LIN {X 0,Y 523.962,Z 330.22,A -85,B 0,C 180,E1 -4900.135,E2 -4900.135} C_VEL
LIN {X 0,Y 523.916,Z 330.218,A -85,B 0,C 180,E1 -4903.168,E2 -4903.168} C_VEL
LIN {X 0,Y 523.936,Z 330.219,A -85,B 0,C 180,E1 -4905.773,E2 -4905.773} C_VEL
LIN {X 0,Y 523.917,Z 330.219,A -85,B 0,C 180,E1 -4906.932,E2 -4906.932} C_VEL
LIN {X 0,Y 523.251,Z 330.304,A -85,B 0,C 180,E1 -4907.573,E2 -4907.573} C_VEL
LIN {X 0,Y 520.406,Z 330.664,A -85,B 0,C 180,E1 -4908.615,E2 -4908.615} C_VEL
LIN {X 0,Y 518,Z 330.967,A -85,B 0,C 180,E1 -4909.454,E2 -4909.454} C_VEL
LIN {X 0,Y 516.963,Z 331.094,A -85,B 0,C 180,E1 -4910.101,E2 -4910.101} C_VEL
LIN {X 0,Y 516.877,Z 331.101,A -85,B 0,C 180,E1 -4910.321,E2 -4910.321} C_VEL
LIN {X 0,Y 516.882,Z 331.095,A -85,B 0,C 180,E1 -4913.343,E2 -4913.343} C_VEL
LIN {X 0,Y 516.909,Z 331.099,A -85,B 0,C 180,E1 -4916.122,E2 -4916.122} C_VEL
LIN {X 0,Y 516.892,Z 331.093,A -85,B 0,C 180,E1 -4918.936,E2 -4918.936} C_VEL
LIN {X 0,Y 516.925,Z 331.093,A -85,B 0,C 180,E1 -4921.586,E2 -4921.586} C_VEL
LIN {X 0,Y 516.934,Z 331.093,A -85,B 0,C 180,E1 -4924.212,E2 -4924.212} C_VEL
LIN {X 0,Y 516.873,Z 331.096,A -85,B 0,C 180,E1 -4926.777,E2 -4926.777} C_VEL
LIN {X 0,Y 516.941,Z 331.095,A -85,B 0,C 180,E1 -4929.732,E2 -4929.732} C_VEL
LIN {X 0,Y 516.931,Z 331.089,A -85,B 0,C 180,E1 -4932.597,E2 -4932.597} C_VEL
LIN {X 0,Y 516.944,Z 331.088,A -85,B 0,C 180,E1 -4935.031,E2 -4935.031} C_VEL
LIN {X 0,Y 516.968,Z 331.086,A -85,B 0,C 180,E1 -4938.234,E2 -4938.234} C_VEL
LIN {X 0,Y 516.973,Z 331.089,A -85,B 0,C 180,E1 -4941.4,E2 -4941.4} C_VEL
LIN {X 0,Y 517.018,Z 331.085,A -85,B 0,C 180,E1 -4943.757,E2 -4943.757} C_VEL
LIN {X 0,Y 517.089,Z 331.077,A -85,B 0,C 180,E1 -4947.663,E2 -4947.663} C_VEL
LIN {X 0,Y 517.097,Z 331.068,A -85,B 0,C 180,E1 -4950.779,E2 -4950.779} C_VEL
LIN {X 0,Y 517.017,Z 331.082,A -85,B 0,C 180,E1 -4953.117,E2 -4953.117} C_VEL
LIN {X 0,Y 517.006,Z 331.08,A -85,B 0,C 180,E1 -4956.243,E2 -4956.243} C_VEL
LIN {X 0,Y 516.955,Z 331.095,A -85,B 0,C 180,E1 -4959.389,E2 -4959.389} C_VEL
LIN {X 0,Y 516.955,Z 331.089,A -85,B 0,C 180,E1 -4961.807,E2 -4961.807} C_VEL
LIN {X 0,Y 516.947,Z 331.093,A -85,B 0,C 180,E1 -4965.146,E2 -4965.146} C_VEL
LIN {X 0,Y 516.928,Z 331.089,A -85,B 0,C 180,E1 -4968.222,E2 -4968.222} C_VEL
LIN {X 0,Y 516.914,Z 331.093,A -85,B 0,C 180,E1 -4970.701,E2 -4970.701} C_VEL
LIN {X 0,Y 516.912,Z 331.091,A -85,B 0,C 180,E1 -4974.071,E2 -4974.071} C_VEL
LIN {X 0,Y 516.93,Z 331.091,A -85,B 0,C 180,E1 -4976.657,E2 -4976.657} C_VEL
LIN {X 0,Y 516.911,Z 331.095,A -85,B 0,C 180,E1 -4979.523,E2 -4979.523} C_VEL
LIN {X 0,Y 516.9,Z 331.094,A -85,B 0,C 180,E1 -4982.544,E2 -4982.544} C_VEL
LIN {X 0,Y 516.882,Z 331.1,A -85,B 0,C 180,E1 -4985.332,E2 -4985.332} C_VEL
LIN {X 0,Y 516.883,Z 331.095,A -85,B 0,C 180,E1 -4987.943,E2 -4987.943} C_VEL
LIN {X 0,Y 516.905,Z 331.099,A -85,B 0,C 180,E1 -4990.738,E2 -4990.738} C_VEL
LIN {X 0,Y 516.879,Z 331.098,A -85,B 0,C 180,E1 -4993.902,E2 -4993.902} C_VEL
LIN {X 0,Y 516.878,Z 331.099,A -85,B 0,C 180,E1 -4996.106,E2 -4996.106} C_VEL
LIN {X 0,Y 516.976,Z 331.211,A -85,B 0,C 180,E1 -4998.813,E2 -4998.813} C_VEL
LIN {X 0,Y 517.149,Z 332.196,A -85,B 0,C 180,E1 -4998.951,E2 -4998.951} C_VEL
LIN {X 0,Y 518.369,Z 337.455,A -85,B 0,C 180,E1 -4999.243,E2 -4999.243} C_VEL
LIN {X 0,Y 518.098,Z 348.894,A -85,B 0,C 180,E1 -4999.884,E2 -4999.884} C_VEL
LIN {X 0,Y 517.795,Z 359.988,A -85,B 0,C 180,E1 -5000.682,E2 -5000.682} C_VEL
LIN {X 0,Y 517.565,Z 369.47,A -85,B 0,C 180,E1 -5001.529,E2 -5001.529} C_VEL
LIN {X 0,Y 517.23,Z 378.856,A -85,B 0,C 180,E1 -5002.551,E2 -5002.551} C_VEL
LIN {X 0,Y 517.051,Z 386.171,A -85,B 0,C 180,E1 -5003.531,E2 -5003.531} C_VEL
LIN {X 0,Y 516.817,Z 393.185,A -85,B 0,C 180,E1 -5004.676,E2 -5004.676} C_VEL
LIN {X 0,Y 516.705,Z 398.028,A -85,B 0,C 180,E1 -5005.635,E2 -5005.635} C_VEL
LIN {X 0,Y 516.538,Z 403.624,A -85,B 0,C 180,E1 -5007.027,E2 -5007.027} C_VEL
LIN {X 0,Y 516.496,Z 407.58,A -85,B 0,C 180,E1 -5008.408,E2 -5008.408} C_VEL
LIN {X 0,Y 516.427,Z 410.24,A -85,B 0,C 180,E1 -5009.766,E2 -5009.766} C_VEL
LIN {X 0,Y 516.38,Z 411.277,A -85,B 0,C 180,E1 -5010.662,E2 -5010.662} C_VEL
LIN {X 0,Y 516.384,Z 411.94,A -85,B 0,C 180,E1 -5012.206,E2 -5012.206} C_VEL
LIN {X 0,Y 516.38,Z 411.461,A -85,B 0,C 180,E1 -5013.312,E2 -5013.312} C_VEL
LIN {X 0,Y 516.426,Z 410.54,A -85,B 0,C 180,E1 -5014.184,E2 -5014.184} C_VEL
LIN {X 0,Y 516.469,Z 409.129,A -85,B 0,C 180,E1 -5015.049,E2 -5015.049} C_VEL
LIN {X 0,Y 516.557,Z 406.079,A -85,B 0,C 180,E1 -5016.337,E2 -5016.337} C_VEL
LIN {X 0,Y 516.692,Z 401.665,A -85,B 0,C 180,E1 -5017.654,E2 -5017.654} C_VEL
LIN {X 0,Y 516.837,Z 395.319,A -85,B 0,C 180,E1 -5019.087,E2 -5019.087} C_VEL
LIN {X 0,Y 517.055,Z 388.019,A -85,B 0,C 180,E1 -5020.342,E2 -5020.342} C_VEL
LIN {X 0,Y 517.297,Z 380.58,A -85,B 0,C 180,E1 -5021.381,E2 -5021.381} C_VEL
LIN {X 0,Y 517.573,Z 371.1,A -85,B 0,C 180,E1 -5022.457,E2 -5022.457} C_VEL
LIN {X 0,Y 517.845,Z 361.431,A -85,B 0,C 180,E1 -5023.339,E2 -5023.339} C_VEL
LIN {X 0,Y 518.133,Z 350.286,A -85,B 0,C 180,E1 -5024.158,E2 -5024.158} C_VEL
LIN {X 0,Y 518.394,Z 338.832,A -85,B 0,C 180,E1 -5024.816,E2 -5024.816} C_VEL
LIN {X 0,Y 518.185,Z 335.842,A -85,B 0,C 180,E1 -5024.968,E2 -5024.968} C_VEL
LIN {X 0,Y 517.053,Z 331.596,A -85,B 0,C 180,E1 -5025.235,E2 -5025.235} C_VEL
LIN {X 0,Y 516.923,Z 331.103,A -85,B 0,C 180,E1 -5025.432,E2 -5025.432} C_VEL
LIN {X 0,Y 516.955,Z 331.09,A -85,B 0,C 180,E1 -5028.233,E2 -5028.233} C_VEL
LIN {X 0,Y 516.958,Z 331.095,A -85,B 0,C 180,E1 -5031.4,E2 -5031.4} C_VEL
LIN {X 0,Y 516.989,Z 331.087,A -85,B 0,C 180,E1 -5033.757,E2 -5033.757} C_VEL
LIN {X 0,Y 517.001,Z 331.085,A -85,B 0,C 180,E1 -5036.883,E2 -5036.883} C_VEL
LIN {X 0,Y 517.068,Z 331.074,A -85,B 0,C 180,E1 -5040,E2 -5040} C_VEL
LIN {X 0,Y 517.002,Z 331.088,A -85,B 0,C 180,E1 -5043.117,E2 -5043.117} C_VEL
LIN {X 0,Y 516.989,Z 331.082,A -85,B 0,C 180,E1 -5046.243,E2 -5046.243} C_VEL
LIN {X 0,Y 516.936,Z 331.094,A -85,B 0,C 180,E1 -5049.39,E2 -5049.39} C_VEL
LIN {X 0,Y 516.941,Z 331.089,A -85,B 0,C 180,E1 -5051.807,E2 -5051.807} C_VEL
LIN {X 0,Y 516.933,Z 331.097,A -85,B 0,C 180,E1 -5055.147,E2 -5055.147} C_VEL
LIN {X 0,Y 516.905,Z 331.091,A -85,B 0,C 180,E1 -5058.223,E2 -5058.223} C_VEL
LIN {X 0,Y 516.901,Z 331.097,A -85,B 0,C 180,E1 -5060.702,E2 -5060.702} C_VEL
LIN {X 0,Y 516.879,Z 331.095,A -85,B 0,C 180,E1 -5064.074,E2 -5064.074} C_VEL
LIN {X 0,Y 516.914,Z 331.096,A -85,B 0,C 180,E1 -5066.659,E2 -5066.659} C_VEL
LIN {X 0,Y 516.899,Z 331.095,A -85,B 0,C 180,E1 -5069.524,E2 -5069.524} C_VEL
LIN {X 0,Y 516.885,Z 331.1,A -85,B 0,C 180,E1 -5072.544,E2 -5072.544} C_VEL
LIN {X 0,Y 516.857,Z 331.102,A -85,B 0,C 180,E1 -5075.33,E2 -5075.33} C_VEL
LIN {X 0,Y 516.871,Z 331.098,A -85,B 0,C 180,E1 -5077.943,E2 -5077.943} C_VEL
LIN {X 0,Y 516.846,Z 331.108,A -85,B 0,C 180,E1 -5080.745,E2 -5080.745} C_VEL
LIN {X 0,Y 516.875,Z 331.098,A -85,B 0,C 180,E1 -5083.904,E2 -5083.904} C_VEL
LIN {X 0,Y 516.875,Z 331.1,A -85,B 0,C 180,E1 -5086.108,E2 -5086.108} C_VEL
LIN {X 0,Y 516.849,Z 331.104,A -85,B 0,C 180,E1 -5089.256,E2 -5089.256} C_VEL
LIN {X 0,Y 516.911,Z 331.323,A -85,B 0,C 180,E1 -5092.053,E2 -5092.053} C_VEL
LIN {X 0,Y 518.241,Z 338.355,A -85,B 0,C 180,E1 -5093.85,E2 -5093.85} C_VEL
LIN {X 0,Y 518.188,Z 344.44,A -85,B 0,C 180,E1 -5095.277,E2 -5095.277} C_VEL
LIN {X 0,Y 517.75,Z 358.665,A -85,B 0,C 180,E1 -5098.45,E2 -5098.45} C_VEL
LIN {X 0,Y 517.637,Z 370.384,A -85,B 0,C 180,E1 -5100.963,E2 -5100.963} C_VEL
LIN {X 0,Y 517.472,Z 384.841,A -85,B 0,C 180,E1 -5103.959,E2 -5103.959} C_VEL
LIN {X 0,Y 517.305,Z 400.935,A -85,B 0,C 180,E1 -5107.195,E2 -5107.195} C_VEL
LIN {X 0,Y 517.105,Z 416.945,A -85,B 0,C 180,E1 -5110.344,E2 -5110.344} C_VEL
LIN {X 0,Y 516.951,Z 430.617,A -85,B 0,C 180,E1 -5113.005,E2 -5113.005} C_VEL
LIN {X 0,Y 516.782,Z 445.74,A -85,B 0,C 180,E1 -5115.931,E2 -5115.931} C_VEL
LIN {X 0,Y 516.772,Z 446.824,A -85,B 0,C 180,E1 -5116.056,E2 -5116.056} C_VEL
LIN {X 0,Y 518.022,Z 457.401,A -85,B 0,C 180,E1 -5116.316,E2 -5116.316} C_VEL
LIN {X 0,Y 518.329,Z 462.091,A -85,B 0,C 180,E1 -5116.449,E2 -5116.449} C_VEL
LIN {X 0,Y 518.085,Z 475.478,A -85,B 0,C 180,E1 -5116.917,E2 -5116.917} C_VEL
LIN {X 0,Y 517.828,Z 488.026,A -85,B 0,C 180,E1 -5117.532,E2 -5117.532} C_VEL
LIN {X 0,Y 517.576,Z 499.386,A -85,B 0,C 180,E1 -5118.248,E2 -5118.248} C_VEL
LIN {X 0,Y 517.292,Z 510.601,A -85,B 0,C 180,E1 -5119.135,E2 -5119.135} C_VEL
LIN {X 0,Y 516.965,Z 519.69,A -85,B 0,C 180,E1 -5120.019,E2 -5120.019} C_VEL
LIN {X 0,Y 516.735,Z 529.581,A -85,B 0,C 180,E1 -5121.199,E2 -5121.199} C_VEL
LIN {X 0,Y 516.563,Z 537.519,A -85,B 0,C 180,E1 -5122.377,E2 -5122.377} C_VEL
LIN {X 0,Y 516.462,Z 543.17,A -85,B 0,C 180,E1 -5123.406,E2 -5123.406} C_VEL
LIN {X 0,Y 516.403,Z 548.195,A -85,B 0,C 180,E1 -5124.533,E2 -5124.533} C_VEL
LIN {X 0,Y 516.36,Z 552.279,A -85,B 0,C 180,E1 -5125.707,E2 -5125.707} C_VEL
LIN {X 0,Y 516.282,Z 555.285,A -85,B 0,C 180,E1 -5126.879,E2 -5126.879} C_VEL
LIN {X 0,Y 516.261,Z 556.726,A -85,B 0,C 180,E1 -5127.659,E2 -5127.659} C_VEL
LIN {X 0,Y 516.162,Z 558.361,A -85,B 0,C 180,E1 -5129.22,E2 -5129.22} C_VEL
LIN {X 0,Y 516.159,Z 558.584,A -85,B 0,C 180,E1 -5130,E2 -5130} C_VEL
LIN {X 0,Y 516.162,Z 558.364,A -85,B 0,C 180,E1 -5130.78,E2 -5130.78} C_VEL
LIN {X 0,Y 516.261,Z 556.735,A -85,B 0,C 180,E1 -5132.341,E2 -5132.341} C_VEL
LIN {X 0,Y 516.282,Z 555.301,A -85,B 0,C 180,E1 -5133.121,E2 -5133.121} C_VEL
LIN {X 0,Y 516.36,Z 552.302,A -85,B 0,C 180,E1 -5134.293,E2 -5134.293} C_VEL
LIN {X 0,Y 516.403,Z 548.232,A -85,B 0,C 180,E1 -5135.467,E2 -5135.467} C_VEL
LIN {X 0,Y 516.483,Z 542.141,A -85,B 0,C 180,E1 -5136.805,E2 -5136.805} C_VEL
LIN {X 0,Y 516.64,Z 535.153,A -85,B 0,C 180,E1 -5138.015,E2 -5138.015} C_VEL
LIN {X 0,Y 516.813,Z 526.702,A -85,B 0,C 180,E1 -5139.194,E2 -5139.194} C_VEL
LIN {X 0,Y 517.04,Z 518.021,A -85,B 0,C 180,E1 -5140.178,E2 -5140.178} C_VEL
LIN {X 0,Y 517.339,Z 507.38,A -85,B 0,C 180,E1 -5141.162,E2 -5141.162} C_VEL
LIN {X 0,Y 517.652,Z 496.773,A -85,B 0,C 180,E1 -5141.956,E2 -5141.956} C_VEL
LIN {X 0,Y 517.883,Z 485.3,A -85,B 0,C 180,E1 -5142.64,E2 -5142.64} C_VEL
LIN {X 0,Y 518.196,Z 472.203,A -85,B 0,C 180,E1 -5143.23,E2 -5143.23} C_VEL
LIN {X 0,Y 518.357,Z 459.09,A -85,B 0,C 180,E1 -5143.65,E2 -5143.65} C_VEL
LIN {X 0,Y 516.789,Z 447.402,A -85,B 0,C 180,E1 -5143.943,E2 -5143.943} C_VEL
LIN {X 0,Y 516.83,Z 445.814,A -85,B 0,C 180,E1 -5144.168,E2 -5144.168} C_VEL
LIN {X 0,Y 516.996,Z 429.457,A -85,B 0,C 180,E1 -5147.401,E2 -5147.401} C_VEL
LIN {X 0,Y 517.162,Z 415.971,A -85,B 0,C 180,E1 -5150.1,E2 -5150.1} C_VEL
LIN {X 0,Y 517.433,Z 402.623,A -85,B 0,C 180,E1 -5152.821,E2 -5152.821} C_VEL
LIN {X 0,Y 517.748,Z 387.104,A -85,B 0,C 180,E1 -5156.064,E2 -5156.064} C_VEL
LIN {X 0,Y 518.026,Z 372.315,A -85,B 0,C 180,E1 -5159.235,E2 -5159.235} C_VEL
LIN {X 0,Y 518.311,Z 360.147,A -85,B 0,C 180,E1 -5161.925,E2 -5161.925} C_VEL
LIN {X 0,Y 518.941,Z 344.977,A -85,B 0,C 180,E1 -5165.376,E2 -5165.376} C_VEL
LIN {X 0,Y 518.836,Z 340.922,A -85,B 0,C 180,E1 -5166.342,E2 -5166.342} C_VEL
LIN {X 0,Y 516.875,Z 331.191,A -85,B 0,C 180,E1 -5168.864,E2 -5168.864} C_VEL
LIN {X 0,Y 516.878,Z 331.103,A -85,B 0,C 180,E1 -5171.777,E2 -5171.777} C_VEL
LIN {X 0,Y 516.89,Z 331.1,A -85,B 0,C 180,E1 -5175.006,E2 -5175.006} C_VEL
LIN {X 0,Y 516.88,Z 331.095,A -85,B 0,C 180,E1 -5178.401,E2 -5178.401} C_VEL
LIN {X 0,Y 516.869,Z 331.105,A -85,B 0,C 180,E1 -5181.283,E2 -5181.283} C_VEL
LIN {X 0,Y 516.862,Z 331.097,A -85,B 0,C 180,E1 -5184.219,E2 -5184.219} C_VEL
LIN {X 0,Y 516.872,Z 331.102,A -85,B 0,C 180,E1 -5187.051,E2 -5187.051} C_VEL
LIN {X 0,Y 516.877,Z 331.097,A -85,B 0,C 180,E1 -5189.795,E2 -5189.795} C_VEL
LIN {X 0,Y 516.915,Z 331.091,A -85,B 0,C 180,E1 -5192.467,E2 -5192.467} C_VEL
LIN {X 0,Y 516.861,Z 331.105,A -85,B 0,C 180,E1 -5195.069,E2 -5195.069} C_VEL
LIN {X 0,Y 516.859,Z 331.1,A -85,B 0,C 180,E1 -5197.621,E2 -5197.621} C_VEL
LIN {X 0,Y 516.92,Z 331.09,A -85,B 0,C 180,E1 -5200.129,E2 -5200.129} C_VEL
LIN {X 0,Y 516.896,Z 331.096,A -85,B 0,C 180,E1 -5202.595,E2 -5202.595} C_VEL
LIN {X 0,Y 516.931,Z 331.098,A -85,B 0,C 180,E1 -5205.03,E2 -5205.03} C_VEL
LIN {X 0,Y 516.955,Z 331.086,A -85,B 0,C 180,E1 -5208.233,E2 -5208.233} C_VEL
LIN {X 0,Y 516.945,Z 331.089,A -85,B 0,C 180,E1 -5211.399,E2 -5211.399} C_VEL
LIN {X 0,Y 516.989,Z 331.081,A -85,B 0,C 180,E1 -5213.757,E2 -5213.757} C_VEL
LIN {X 0,Y 517.001,Z 331.089,A -85,B 0,C 180,E1 -5216.883,E2 -5216.883} C_VEL
LIN {X 0,Y 517.068,Z 331.072,A -85,B 0,C 180,E1 -5220,E2 -5220} C_VEL
LIN {X 0,Y 517.001,Z 331.084,A -85,B 0,C 180,E1 -5223.117,E2 -5223.117} C_VEL
LIN {X 0,Y 516.989,Z 331.084,A -85,B 0,C 180,E1 -5226.243,E2 -5226.243} C_VEL
LIN {X 0,Y 516.943,Z 331.088,A -85,B 0,C 180,E1 -5229.389,E2 -5229.389} C_VEL
LIN {X 0,Y 516.943,Z 331.087,A -85,B 0,C 180,E1 -5231.808,E2 -5231.808} C_VEL
LIN {X 0,Y 516.936,Z 331.09,A -85,B 0,C 180,E1 -5235.148,E2 -5235.148} C_VEL
LIN {X 0,Y 516.915,Z 331.095,A -85,B 0,C 180,E1 -5238.223,E2 -5238.223} C_VEL
LIN {X 0,Y 516.906,Z 331.098,A -85,B 0,C 180,E1 -5240.702,E2 -5240.702} C_VEL
LIN {X 0,Y 516.883,Z 331.095,A -85,B 0,C 180,E1 -5243.223,E2 -5243.223} C_VEL
LIN {X 0,Y 516.934,Z 331.094,A -85,B 0,C 180,E1 -5246.197,E2 -5246.197} C_VEL
LIN {X 0,Y 516.928,Z 331.089,A -85,B 0,C 180,E1 -5249.304,E2 -5249.304} C_VEL
LIN {X 0,Y 516.889,Z 331.1,A -85,B 0,C 180,E1 -5252.544,E2 -5252.544} C_VEL
LIN {X 0,Y 516.872,Z 331.096,A -85,B 0,C 180,E1 -5255.332,E2 -5255.332} C_VEL
LIN {X 0,Y 516.874,Z 331.1,A -85,B 0,C 180,E1 -5257.944,E2 -5257.944} C_VEL
LIN {X 0,Y 516.898,Z 331.095,A -85,B 0,C 180,E1 -5260.74,E2 -5260.74} C_VEL
LIN {X 0,Y 516.877,Z 331.1,A -85,B 0,C 180,E1 -5263.904,E2 -5263.904} C_VEL
LIN {X 0,Y 516.878,Z 331.104,A -85,B 0,C 180,E1 -5266.108,E2 -5266.108} C_VEL
LIN {X 0,Y 516.911,Z 331.096,A -85,B 0,C 180,E1 -5268.399,E2 -5268.399} C_VEL
LIN {X 0,Y 516.877,Z 331.101,A -85,B 0,C 180,E1 -5270.321,E2 -5270.321} C_VEL
LIN {X 0,Y 516.207,Z 331.181,A -85,B 0,C 180,E1 -5270.971,E2 -5270.971} C_VEL
LIN {X 0,Y 513.361,Z 331.542,A -85,B 0,C 180,E1 -5272.027,E2 -5272.027} C_VEL
LIN {X 0,Y 510.954,Z 331.841,A -85,B 0,C 180,E1 -5272.877,E2 -5272.877} C_VEL
LIN {X 0,Y 509.915,Z 331.966,A -85,B 0,C 180,E1 -5273.534,E2 -5273.534} C_VEL
LIN {X 0,Y 509.827,Z 331.976,A -85,B 0,C 180,E1 -5273.756,E2 -5273.756} C_VEL
LIN {X 0,Y 509.859,Z 331.972,A -85,B 0,C 180,E1 -5276.54,E2 -5276.54} C_VEL
LIN {X 0,Y 509.849,Z 331.972,A -85,B 0,C 180,E1 -5279.335,E2 -5279.335} C_VEL
LIN {X 0,Y 509.896,Z 331.972,A -85,B 0,C 180,E1 -5282.055,E2 -5282.055} C_VEL
LIN {X 0,Y 509.879,Z 331.967,A -85,B 0,C 180,E1 -5284.705,E2 -5284.705} C_VEL
LIN {X 0,Y 509.837,Z 331.976,A -85,B 0,C 180,E1 -5287.456,E2 -5287.456} C_VEL
LIN {X 0,Y 509.918,Z 331.971,A -85,B 0,C 180,E1 -5289.845,E2 -5289.845} C_VEL
LIN {X 0,Y 509.887,Z 331.968,A -85,B 0,C 180,E1 -5293.175,E2 -5293.175} C_VEL
LIN {X 0,Y 509.867,Z 331.976,A -85,B 0,C 180,E1 -5295.635,E2 -5295.635} C_VEL
LIN {X 0,Y 509.916,Z 331.963,A -85,B 0,C 180,E1 -5298.875,E2 -5298.875} C_VEL
LIN {X 0,Y 509.955,Z 331.961,A -85,B 0,C 180,E1 -5302.079,E2 -5302.079} C_VEL
LIN {X 0,Y 509.988,Z 331.954,A -85,B 0,C 180,E1 -5304.465,E2 -5304.465} C_VEL
LIN {X 0,Y 510.059,Z 331.953,A -85,B 0,C 180,E1 -5307.631,E2 -5307.631} C_VEL
LIN {X 0,Y 510.067,Z 331.944,A -85,B 0,C 180,E1 -5310.789,E2 -5310.789} C_VEL
LIN {X 0,Y 509.959,Z 331.961,A -85,B 0,C 180,E1 -5313.16,E2 -5313.16} C_VEL
LIN {X 0,Y 509.957,Z 331.957,A -85,B 0,C 180,E1 -5316.33,E2 -5316.33} C_VEL
LIN {X 0,Y 509.918,Z 331.963,A -85,B 0,C 180,E1 -5318.72,E2 -5318.72} C_VEL
LIN {X 0,Y 509.907,Z 331.965,A -85,B 0,C 180,E1 -5321.931,E2 -5321.931} C_VEL
LIN {X 0,Y 509.896,Z 331.973,A -85,B 0,C 180,E1 -5325.241,E2 -5325.241} C_VEL
LIN {X 0,Y 509.891,Z 331.966,A -85,B 0,C 180,E1 -5328.001,E2 -5328.001} C_VEL
LIN {X 0,Y 509.852,Z 331.976,A -85,B 0,C 180,E1 -5331.001,E2 -5331.001} C_VEL
LIN {X 0,Y 509.838,Z 331.976,A -85,B 0,C 180,E1 -5333.562,E2 -5333.562} C_VEL
LIN {X 0,Y 509.914,Z 331.963,A -85,B 0,C 180,E1 -5336.379,E2 -5336.379} C_VEL
LIN {X 0,Y 509.877,Z 331.972,A -85,B 0,C 180,E1 -5338.843,E2 -5338.843} C_VEL
LIN {X 0,Y 509.824,Z 331.976,A -85,B 0,C 180,E1 -5341.589,E2 -5341.589} C_VEL
LIN {X 0,Y 509.853,Z 331.971,A -85,B 0,C 180,E1 -5344.412,E2 -5344.412} C_VEL
LIN {X 0,Y 509.821,Z 331.979,A -85,B 0,C 180,E1 -5347.339,E2 -5347.339} C_VEL
LIN {X 0,Y 509.86,Z 331.973,A -85,B 0,C 180,E1 -5350.379,E2 -5350.379} C_VEL
LIN {X 0,Y 509.837,Z 331.98,A -85,B 0,C 180,E1 -5353.064,E2 -5353.064} C_VEL
LIN {X 0,Y 509.826,Z 331.977,A -85,B 0,C 180,E1 -5355.791,E2 -5355.791} C_VEL
LIN {X 0,Y 509.921,Z 332.178,A -85,B 0,C 180,E1 -5358.649,E2 -5358.649} C_VEL
LIN {X 0,Y 510.142,Z 333.081,A -85,B 0,C 180,E1 -5358.772,E2 -5358.772} C_VEL
LIN {X 0,Y 511.495,Z 338.635,A -85,B 0,C 180,E1 -5359.085,E2 -5359.085} C_VEL
LIN {X 0,Y 511.202,Z 350.173,A -85,B 0,C 180,E1 -5359.747,E2 -5359.747} C_VEL
LIN {X 0,Y 510.893,Z 361.197,A -85,B 0,C 180,E1 -5360.555,E2 -5360.555} C_VEL
LIN {X 0,Y 510.59,Z 371.747,A -85,B 0,C 180,E1 -5361.524,E2 -5361.524} C_VEL
LIN {X 0,Y 510.244,Z 381.905,A -85,B 0,C 180,E1 -5362.696,E2 -5362.696} C_VEL
LIN {X 0,Y 510.001,Z 390.072,A -85,B 0,C 180,E1 -5363.874,E2 -5363.874} C_VEL
LIN {X 0,Y 509.798,Z 396.88,A -85,B 0,C 180,E1 -5365.102,E2 -5365.102} C_VEL
LIN {X 0,Y 509.638,Z 401.649,A -85,B 0,C 180,E1 -5366.172,E2 -5366.172} C_VEL
LIN {X 0,Y 509.491,Z 406.118,A -85,B 0,C 180,E1 -5367.454,E2 -5367.454} C_VEL
LIN {X 0,Y 509.457,Z 409.548,A -85,B 0,C 180,E1 -5368.79,E2 -5368.79} C_VEL
LIN {X 0,Y 509.374,Z 411.996,A -85,B 0,C 180,E1 -5370.367,E2 -5370.367} C_VEL
LIN {X 0,Y 509.358,Z 412.662,A -85,B 0,C 180,E1 -5371.124,E2 -5371.124} C_VEL
LIN {X 0,Y 509.351,Z 412.963,A -85,B 0,C 180,E1 -5372.022,E2 -5372.022} C_VEL
LIN {X 0,Y 509.364,Z 412.736,A -85,B 0,C 180,E1 -5372.914,E2 -5372.914} C_VEL
LIN {X 0,Y 509.381,Z 412.029,A -85,B 0,C 180,E1 -5373.8,E2 -5373.8} C_VEL
LIN {X 0,Y 509.433,Z 410.842,A -85,B 0,C 180,E1 -5374.68,E2 -5374.68} C_VEL
LIN {X 0,Y 509.545,Z 408.16,A -85,B 0,C 180,E1 -5375.991,E2 -5375.991} C_VEL
LIN {X 0,Y 509.671,Z 403.589,A -85,B 0,C 180,E1 -5377.497,E2 -5377.497} C_VEL
LIN {X 0,Y 509.794,Z 399.236,A -85,B 0,C 180,E1 -5378.572,E2 -5378.572} C_VEL
LIN {X 0,Y 509.987,Z 392.761,A -85,B 0,C 180,E1 -5379.848,E2 -5379.848} C_VEL
LIN {X 0,Y 510.265,Z 384.563,A -85,B 0,C 180,E1 -5381.115,E2 -5381.115} C_VEL
LIN {X 0,Y 510.578,Z 375.533,A -85,B 0,C 180,E1 -5382.232,E2 -5382.232} C_VEL
LIN {X 0,Y 510.881,Z 365.729,A -85,B 0,C 180,E1 -5383.209,E2 -5383.209} C_VEL
LIN {X 0,Y 511.193,Z 355.362,A -85,B 0,C 180,E1 -5384.04,E2 -5384.04} C_VEL
LIN {X 0,Y 511.496,Z 344.492,A -85,B 0,C 180,E1 -5384.737,E2 -5384.737} C_VEL
LIN {X 0,Y 511.492,Z 338.239,A -85,B 0,C 180,E1 -5385.071,E2 -5385.071} C_VEL
LIN {X 0,Y 510.002,Z 332.602,A -85,B 0,C 180,E1 -5385.409,E2 -5385.409} C_VEL
LIN {X 0,Y 509.871,Z 331.979,A -85,B 0,C 180,E1 -5385.634,E2 -5385.634} C_VEL
LIN {X 0,Y 509.906,Z 331.97,A -85,B 0,C 180,E1 -5388.874,E2 -5388.874} C_VEL
LIN {X 0,Y 509.94,Z 331.963,A -85,B 0,C 180,E1 -5392.078,E2 -5392.078} C_VEL
LIN {X 0,Y 509.967,Z 331.958,A -85,B 0,C 180,E1 -5394.464,E2 -5394.464} C_VEL
LIN {X 0,Y 510.041,Z 331.953,A -85,B 0,C 180,E1 -5397.631,E2 -5397.631} C_VEL
LIN {X 0,Y 510.04,Z 331.95,A -85,B 0,C 180,E1 -5400,E2 -5400} C_VEL
LIN {X 0,Y 510.039,Z 331.948,A -85,B 0,C 180,E1 -5402.369,E2 -5402.369} C_VEL
LIN {X 0,Y 509.966,Z 331.962,A -85,B 0,C 180,E1 -5405.536,E2 -5405.536} C_VEL
LIN {X 0,Y 509.909,Z 331.964,A -85,B 0,C 180,E1 -5407.922,E2 -5407.922} C_VEL
LIN {X 0,Y 509.901,Z 331.974,A -85,B 0,C 180,E1 -5411.126,E2 -5411.126} C_VEL
LIN {X 0,Y 509.851,Z 331.972,A -85,B 0,C 180,E1 -5414.366,E2 -5414.366} C_VEL
LIN {X 0,Y 509.863,Z 331.976,A -85,B 0,C 180,E1 -5416.826,E2 -5416.826} C_VEL
LIN {X 0,Y 509.906,Z 331.964,A -85,B 0,C 180,E1 -5420.156,E2 -5420.156} C_VEL
LIN {X 0,Y 509.81,Z 331.977,A -85,B 0,C 180,E1 -5423.565,E2 -5423.565} C_VEL
LIN {X 0,Y 509.901,Z 331.966,A -85,B 0,C 180,E1 -5426.379,E2 -5426.379} C_VEL
LIN {X 0,Y 509.863,Z 331.976,A -85,B 0,C 180,E1 -5428.845,E2 -5428.845} C_VEL
LIN {X 0,Y 509.809,Z 331.978,A -85,B 0,C 180,E1 -5431.591,E2 -5431.591} C_VEL
LIN {X 0,Y 509.83,Z 331.978,A -85,B 0,C 180,E1 -5434.415,E2 -5434.415} C_VEL
LIN {X 0,Y 509.808,Z 331.98,A -85,B 0,C 180,E1 -5437.342,E2 -5437.342} C_VEL
LIN {X 0,Y 509.807,Z 331.982,A -85,B 0,C 180,E1 -5440.385,E2 -5440.385} C_VEL
LIN {X 0,Y 509.789,Z 331.985,A -85,B 0,C 180,E1 -5443.06,E2 -5443.06} C_VEL
LIN {X 0,Y 509.816,Z 331.978,A -85,B 0,C 180,E1 -5445.794,E2 -5445.794} C_VEL
LIN {X 0,Y 509.826,Z 331.982,A -85,B 0,C 180,E1 -5448.573,E2 -5448.573} C_VEL
LIN {X 0,Y 509.85,Z 332.132,A -85,B 0,C 180,E1 -5451.787,E2 -5451.787} C_VEL
LIN {X 0,Y 511.288,Z 339.689,A -85,B 0,C 180,E1 -5453.769,E2 -5453.769} C_VEL
LIN {X 0,Y 511.253,Z 345.707,A -85,B 0,C 180,E1 -5455.207,E2 -5455.207} C_VEL
LIN {X 0,Y 510.76,Z 360.437,A -85,B 0,C 180,E1 -5458.552,E2 -5458.552} C_VEL
LIN {X 0,Y 510.6,Z 371.564,A -85,B 0,C 180,E1 -5460.976,E2 -5460.976} C_VEL
LIN {X 0,Y 510.422,Z 385.228,A -85,B 0,C 180,E1 -5463.858,E2 -5463.858} C_VEL
LIN {X 0,Y 510.24,Z 401.062,A -85,B 0,C 180,E1 -5467.101,E2 -5467.101} C_VEL
LIN {X 0,Y 510.012,Z 416.878,A -85,B 0,C 180,E1 -5470.269,E2 -5470.269} C_VEL
LIN {X 0,Y 509.871,Z 430.533,A -85,B 0,C 180,E1 -5472.968,E2 -5472.968} C_VEL
LIN {X 0,Y 509.722,Z 445.31,A -85,B 0,C 180,E1 -5475.834,E2 -5475.834} C_VEL
LIN {X 0,Y 509.904,Z 448.112,A -85,B 0,C 180,E1 -5475.928,E2 -5475.928} C_VEL
LIN {X 0,Y 511.065,Z 458.131,A -85,B 0,C 180,E1 -5476.177,E2 -5476.177} C_VEL
LIN {X 0,Y 511.361,Z 463.388,A -85,B 0,C 180,E1 -5476.337,E2 -5476.337} C_VEL
LIN {X 0,Y 511.066,Z 476.455,A -85,B 0,C 180,E1 -5476.835,E2 -5476.835} C_VEL
LIN {X 0,Y 510.784,Z 488.569,A -85,B 0,C 180,E1 -5477.459,E2 -5477.459} C_VEL
LIN {X 0,Y 510.528,Z 499.598,A -85,B 0,C 180,E1 -5478.184,E2 -5478.184} C_VEL
LIN {X 0,Y 510.21,Z 510.505,A -85,B 0,C 180,E1 -5479.082,E2 -5479.082} C_VEL
LIN {X 0,Y 509.876,Z 520.348,A -85,B 0,C 180,E1 -5480.079,E2 -5480.079} C_VEL
LIN {X 0,Y 509.675,Z 528.458,A -85,B 0,C 180,E1 -5481.076,E2 -5481.076} C_VEL
LIN {X 0,Y 509.513,Z 536.424,A -85,B 0,C 180,E1 -5482.271,E2 -5482.271} C_VEL
LIN {X 0,Y 509.367,Z 543.727,A -85,B 0,C 180,E1 -5483.663,E2 -5483.663} C_VEL
LIN {X 0,Y 509.294,Z 548.604,A -85,B 0,C 180,E1 -5484.854,E2 -5484.854} C_VEL
LIN {X 0,Y 509.336,Z 552.348,A -85,B 0,C 180,E1 -5486.044,E2 -5486.044} C_VEL
LIN {X 0,Y 509.243,Z 554.261,A -85,B 0,C 180,E1 -5486.836,E2 -5486.836} C_VEL
LIN {X 0,Y 509.222,Z 555.711,A -85,B 0,C 180,E1 -5487.627,E2 -5487.627} C_VEL
LIN {X 0,Y 509.156,Z 557.366,A -85,B 0,C 180,E1 -5489.209,E2 -5489.209} C_VEL
LIN {X 0,Y 509.149,Z 557.594,A -85,B 0,C 180,E1 -5490,E2 -5490} C_VEL
LIN {X 0,Y 509.156,Z 557.379,A -85,B 0,C 180,E1 -5490.791,E2 -5490.791} C_VEL
LIN {X 0,Y 509.218,Z 555.753,A -85,B 0,C 180,E1 -5492.373,E2 -5492.373} C_VEL
LIN {X 0,Y 509.237,Z 554.319,A -85,B 0,C 180,E1 -5493.164,E2 -5493.164} C_VEL
LIN {X 0,Y 509.282,Z 551.319,A -85,B 0,C 180,E1 -5494.353,E2 -5494.353} C_VEL
LIN {X 0,Y 509.342,Z 547.251,A -85,B 0,C 180,E1 -5495.543,E2 -5495.543} C_VEL
LIN {X 0,Y 509.415,Z 541.338,A -85,B 0,C 180,E1 -5496.864,E2 -5496.864} C_VEL
LIN {X 0,Y 509.571,Z 534.166,A -85,B 0,C 180,E1 -5498.127,E2 -5498.127} C_VEL
LIN {X 0,Y 509.758,Z 525.708,A -85,B 0,C 180,E1 -5499.323,E2 -5499.323} C_VEL
LIN {X 0,Y 510.009,Z 517.023,A -85,B 0,C 180,E1 -5500.32,E2 -5500.32} C_VEL
LIN {X 0,Y 510.298,Z 506.373,A -85,B 0,C 180,E1 -5501.318,E2 -5501.318} C_VEL
LIN {X 0,Y 510.618,Z 495.923,A -85,B 0,C 180,E1 -5502.112,E2 -5502.112} C_VEL
LIN {X 0,Y 510.909,Z 484.279,A -85,B 0,C 180,E1 -5502.815,E2 -5502.815} C_VEL
LIN {X 0,Y 511.274,Z 471.177,A -85,B 0,C 180,E1 -5503.412,E2 -5503.412} C_VEL
LIN {X 0,Y 511.298,Z 459.401,A -85,B 0,C 180,E1 -5503.804,E2 -5503.804} C_VEL
LIN {X 0,Y 509.774,Z 447.382,A -85,B 0,C 180,E1 -5504.113,E2 -5504.113} C_VEL
LIN {X 0,Y 509.75,Z 445.928,A -85,B 0,C 180,E1 -5504.19,E2 -5504.19} C_VEL
LIN {X 0,Y 509.91,Z 430.664,A -85,B 0,C 180,E1 -5507.237,E2 -5507.237} C_VEL
LIN {X 0,Y 510.085,Z 417.396,A -85,B 0,C 180,E1 -5509.938,E2 -5509.938} C_VEL
LIN {X 0,Y 510.372,Z 404.121,A -85,B 0,C 180,E1 -5512.688,E2 -5512.688} C_VEL
LIN {X 0,Y 510.689,Z 388.957,A -85,B 0,C 180,E1 -5515.908,E2 -5515.908} C_VEL
LIN {X 0,Y 511.01,Z 374.729,A -85,B 0,C 180,E1 -5518.998,E2 -5518.998} C_VEL
LIN {X 0,Y 511.349,Z 361.565,A -85,B 0,C 180,E1 -5521.946,E2 -5521.946} C_VEL
LIN {X 0,Y 511.967,Z 347.435,A -85,B 0,C 180,E1 -5525.207,E2 -5525.207} C_VEL
LIN {X 0,Y 512.052,Z 343.388,A -85,B 0,C 180,E1 -5526.169,E2 -5526.169} C_VEL
LIN {X 0,Y 510.072,Z 333.104,A -85,B 0,C 180,E1 -5528.822,E2 -5528.822} C_VEL
LIN {X 0,Y 509.847,Z 332.053,A -85,B 0,C 180,E1 -5529.16,E2 -5529.16} C_VEL
LIN {X 0,Y 509.825,Z 331.981,A -85,B 0,C 180,E1 -5531.892,E2 -5531.892} C_VEL
LIN {X 0,Y 509.833,Z 331.976,A -85,B 0,C 180,E1 -5534.669,E2 -5534.669} C_VEL
LIN {X 0,Y 509.795,Z 331.985,A -85,B 0,C 180,E1 -5537.506,E2 -5537.506} C_VEL
LIN {X 0,Y 509.825,Z 331.975,A -85,B 0,C 180,E1 -5540.645,E2 -5540.645} C_VEL
LIN {X 0,Y 509.817,Z 331.979,A -85,B 0,C 180,E1 -5543.646,E2 -5543.646} C_VEL
LIN {X 0,Y 509.833,Z 331.973,A -85,B 0,C 180,E1 -5546.537,E2 -5546.537} C_VEL
LIN {X 0,Y 509.833,Z 331.98,A -85,B 0,C 180,E1 -5549.333,E2 -5549.333} C_VEL
LIN {X 0,Y 509.88,Z 331.967,A -85,B 0,C 180,E1 -5552.054,E2 -5552.054} C_VEL
LIN {X 0,Y 509.827,Z 331.976,A -85,B 0,C 180,E1 -5554.701,E2 -5554.701} C_VEL
LIN {X 0,Y 509.815,Z 331.979,A -85,B 0,C 180,E1 -5557.458,E2 -5557.458} C_VEL
LIN {X 0,Y 509.906,Z 331.964,A -85,B 0,C 180,E1 -5559.844,E2 -5559.844} C_VEL
LIN {X 0,Y 509.863,Z 331.976,A -85,B 0,C 180,E1 -5563.174,E2 -5563.174} C_VEL
LIN {X 0,Y 509.851,Z 331.972,A -85,B 0,C 180,E1 -5565.634,E2 -5565.634} C_VEL
LIN {X 0,Y 509.901,Z 331.972,A -85,B 0,C 180,E1 -5568.874,E2 -5568.874} C_VEL
LIN {X 0,Y 509.909,Z 331.964,A -85,B 0,C 180,E1 -5572.078,E2 -5572.078} C_VEL
LIN {X 0,Y 509.966,Z 331.959,A -85,B 0,C 180,E1 -5574.464,E2 -5574.464} C_VEL
LIN {X 0,Y 510.039,Z 331.947,A -85,B 0,C 180,E1 -5577.631,E2 -5577.631} C_VEL
LIN {X 0,Y 510.054,Z 331.955,A -85,B 0,C 180,E1 -5580.789,E2 -5580.789} C_VEL
LIN {X 0,Y 509.943,Z 331.962,A -85,B 0,C 180,E1 -5583.16,E2 -5583.16} C_VEL
LIN {X 0,Y 509.941,Z 331.963,A -85,B 0,C 180,E1 -5586.33,E2 -5586.33} C_VEL
LIN {X 0,Y 509.905,Z 331.973,A -85,B 0,C 180,E1 -5588.72,E2 -5588.72} C_VEL
LIN {X 0,Y 509.894,Z 331.966,A -85,B 0,C 180,E1 -5591.932,E2 -5591.932} C_VEL
LIN {X 0,Y 509.883,Z 331.968,A -85,B 0,C 180,E1 -5595.242,E2 -5595.242} C_VEL
LIN {X 0,Y 509.878,Z 331.969,A -85,B 0,C 180,E1 -5598.001,E2 -5598.001} C_VEL
LIN {X 0,Y 509.848,Z 331.973,A -85,B 0,C 180,E1 -5601.002,E2 -5601.002} C_VEL
LIN {X 0,Y 509.841,Z 331.972,A -85,B 0,C 180,E1 -5603.563,E2 -5603.563} C_VEL
LIN {X 0,Y 509.903,Z 331.973,A -85,B 0,C 180,E1 -5606.379,E2 -5606.379} C_VEL
LIN {X 0,Y 509.877,Z 331.97,A -85,B 0,C 180,E1 -5608.844,E2 -5608.844} C_VEL
LIN {X 0,Y 509.814,Z 331.976,A -85,B 0,C 180,E1 -5611.591,E2 -5611.591} C_VEL
LIN {X 0,Y 509.844,Z 331.979,A -85,B 0,C 180,E1 -5614.414,E2 -5614.414} C_VEL
LIN {X 0,Y 509.812,Z 331.975,A -85,B 0,C 180,E1 -5617.341,E2 -5617.341} C_VEL
LIN {X 0,Y 509.854,Z 331.977,A -85,B 0,C 180,E1 -5620.381,E2 -5620.381} C_VEL
LIN {X 0,Y 509.818,Z 331.975,A -85,B 0,C 180,E1 -5623.063,E2 -5623.063} C_VEL
LIN {X 0,Y 509.826,Z 331.977,A -85,B 0,C 180,E1 -5625.793,E2 -5625.793} C_VEL
LIN {X 0,Y 509.853,Z 331.973,A -85,B 0,C 180,E1 -5628.576,E2 -5628.576} C_VEL
LIN {X 0,Y 509.848,Z 331.976,A -85,B 0,C 180,E1 -5631.787,E2 -5631.787} C_VEL
LIN {X 0,Y 509.827,Z 331.976,A -85,B 0,C 180,E1 -5633.756,E2 -5633.756} C_VEL
LIN {X 0,Y 509.162,Z 332.06,A -85,B 0,C 180,E1 -5634.416,E2 -5634.416} C_VEL
LIN {X 0,Y 506.344,Z 332.409,A -85,B 0,C 180,E1 -5635.488,E2 -5635.488} C_VEL
LIN {X 0,Y 503.951,Z 332.71,A -85,B 0,C 180,E1 -5636.351,E2 -5636.351} C_VEL
LIN {X 0,Y 502.902,Z 332.837,A -85,B 0,C 180,E1 -5637.017,E2 -5637.017} C_VEL
LIN {X 0,Y 502.805,Z 332.849,A -85,B 0,C 180,E1 -5637.243,E2 -5637.243} C_VEL
LIN {X 0,Y 502.83,Z 332.853,A -85,B 0,C 180,E1 -5640.062,E2 -5640.062} C_VEL
LIN {X 0,Y 502.836,Z 332.846,A -85,B 0,C 180,E1 -5642.534,E2 -5642.534} C_VEL
LIN {X 0,Y 502.83,Z 332.847,A -85,B 0,C 180,E1 -5645.299,E2 -5645.299} C_VEL
LIN {X 0,Y 502.786,Z 332.859,A -85,B 0,C 180,E1 -5647.827,E2 -5647.827} C_VEL
LIN {X 0,Y 502.826,Z 332.847,A -85,B 0,C 180,E1 -5650.401,E2 -5650.401} C_VEL
LIN {X 0,Y 502.836,Z 332.845,A -85,B 0,C 180,E1 -5652.932,E2 -5652.932} C_VEL
LIN {X 0,Y 502.847,Z 332.847,A -85,B 0,C 180,E1 -5655.43,E2 -5655.43} C_VEL
LIN {X 0,Y 502.88,Z 332.839,A -85,B 0,C 180,E1 -5658.717,E2 -5658.717} C_VEL
LIN {X 0,Y 502.905,Z 332.84,A -85,B 0,C 180,E1 -5661.967,E2 -5661.967} C_VEL
LIN {X 0,Y 502.944,Z 332.831,A -85,B 0,C 180,E1 -5664.387,E2 -5664.387} C_VEL
LIN {X 0,Y 503.029,Z 332.829,A -85,B 0,C 180,E1 -5667.598,E2 -5667.598} C_VEL
LIN {X 0,Y 503.031,Z 332.823,A -85,B 0,C 180,E1 -5670,E2 -5670} C_VEL
LIN {X 0,Y 503.029,Z 332.821,A -85,B 0,C 180,E1 -5672.402,E2 -5672.402} C_VEL
LIN {X 0,Y 502.937,Z 332.839,A -85,B 0,C 180,E1 -5675.613,E2 -5675.613} C_VEL
LIN {X 0,Y 502.905,Z 332.837,A -85,B 0,C 180,E1 -5678.033,E2 -5678.033} C_VEL
LIN {X 0,Y 502.88,Z 332.846,A -85,B 0,C 180,E1 -5681.283,E2 -5681.283} C_VEL
LIN {X 0,Y 502.848,Z 332.844,A -85,B 0,C 180,E1 -5684.57,E2 -5684.57} C_VEL
LIN {X 0,Y 502.864,Z 332.842,A -85,B 0,C 180,E1 -5687.906,E2 -5687.906} C_VEL
LIN {X 0,Y 502.83,Z 332.846,A -85,B 0,C 180,E1 -5690.536,E2 -5690.536} C_VEL
LIN {X 0,Y 502.798,Z 332.855,A -85,B 0,C 180,E1 -5693.04,E2 -5693.04} C_VEL
LIN {X 0,Y 502.842,Z 332.846,A -85,B 0,C 180,E1 -5695.675,E2 -5695.675} C_VEL
LIN {X 0,Y 502.84,Z 332.844,A -85,B 0,C 180,E1 -5698.372,E2 -5698.372} C_VEL
LIN {X 0,Y 502.795,Z 332.853,A -85,B 0,C 180,E1 -5701.499,E2 -5701.499} C_VEL
LIN {X 0,Y 502.806,Z 332.85,A -85,B 0,C 180,E1 -5704.444,E2 -5704.444} C_VEL
LIN {X 0,Y 502.782,Z 332.858,A -85,B 0,C 180,E1 -5707.178,E2 -5707.178} C_VEL
LIN {X 0,Y 502.824,Z 332.848,A -85,B 0,C 180,E1 -5710.011,E2 -5710.011} C_VEL
LIN {X 0,Y 502.823,Z 332.849,A -85,B 0,C 180,E1 -5712.201,E2 -5712.201} C_VEL
LIN {X 0,Y 502.796,Z 332.855,A -85,B 0,C 180,E1 -5715.467,E2 -5715.467} C_VEL
LIN {X 0,Y 502.891,Z 333.063,A -85,B 0,C 180,E1 -5718.464,E2 -5718.464} C_VEL
LIN {X 0,Y 503.087,Z 334.039,A -85,B 0,C 180,E1 -5718.589,E2 -5718.589} C_VEL
LIN {X 0,Y 504.588,Z 340.032,A -85,B 0,C 180,E1 -5718.936,E2 -5718.936} C_VEL
LIN {X 0,Y 504.329,Z 352.254,A -85,B 0,C 180,E1 -5719.662,E2 -5719.662} C_VEL
LIN {X 0,Y 503.947,Z 363.121,A -85,B 0,C 180,E1 -5720.485,E2 -5720.485} C_VEL
LIN {X 0,Y 503.631,Z 373.513,A -85,B 0,C 180,E1 -5721.472,E2 -5721.472} C_VEL
LIN {X 0,Y 503.333,Z 382.341,A -85,B 0,C 180,E1 -5722.505,E2 -5722.505} C_VEL
LIN {X 0,Y 503.052,Z 389.833,A -85,B 0,C 180,E1 -5723.576,E2 -5723.576} C_VEL
LIN {X 0,Y 502.855,Z 396.855,A -85,B 0,C 180,E1 -5724.812,E2 -5724.812} C_VEL
LIN {X 0,Y 502.67,Z 402.219,A -85,B 0,C 180,E1 -5725.996,E2 -5725.996} C_VEL
LIN {X 0,Y 502.516,Z 406.049,A -85,B 0,C 180,E1 -5727.047,E2 -5727.047} C_VEL
LIN {X 0,Y 502.467,Z 410.11,A -85,B 0,C 180,E1 -5728.56,E2 -5728.56} C_VEL
LIN {X 0,Y 502.379,Z 412.8,A -85,B 0,C 180,E1 -5730.149,E2 -5730.149} C_VEL
LIN {X 0,Y 502.321,Z 413.918,A -85,B 0,C 180,E1 -5731.813,E2 -5731.813} C_VEL
LIN {X 0,Y 502.345,Z 413.902,A -85,B 0,C 180,E1 -5732.504,E2 -5732.504} C_VEL
LIN {X 0,Y 502.364,Z 413.302,A -85,B 0,C 180,E1 -5733.551,E2 -5733.551} C_VEL
LIN {X 0,Y 502.396,Z 412.486,A -85,B 0,C 180,E1 -5734.3,E2 -5734.3} C_VEL
LIN {X 0,Y 502.476,Z 410.667,A -85,B 0,C 180,E1 -5735.383,E2 -5735.383} C_VEL
LIN {X 0,Y 502.65,Z 406.66,A -85,B 0,C 180,E1 -5736.953,E2 -5736.953} C_VEL
LIN {X 0,Y 502.793,Z 401.996,A -85,B 0,C 180,E1 -5738.259,E2 -5738.259} C_VEL
LIN {X 0,Y 502.97,Z 395.943,A -85,B 0,C 180,E1 -5739.554,E2 -5739.554} C_VEL
LIN {X 0,Y 503.248,Z 388.336,A -85,B 0,C 180,E1 -5740.841,E2 -5740.841} C_VEL
LIN {X 0,Y 503.525,Z 380.099,A -85,B 0,C 180,E1 -5741.958,E2 -5741.958} C_VEL
LIN {X 0,Y 503.896,Z 369.818,A -85,B 0,C 180,E1 -5743.073,E2 -5743.073} C_VEL
LIN {X 0,Y 504.205,Z 359.82,A -85,B 0,C 180,E1 -5743.948,E2 -5743.948} C_VEL
LIN {X 0,Y 504.523,Z 348.107,A -85,B 0,C 180,E1 -5744.756,E2 -5744.756} C_VEL
LIN {X 0,Y 504.708,Z 340.658,A -85,B 0,C 180,E1 -5745.175,E2 -5745.175} C_VEL
LIN {X 0,Y 503.596,Z 335.789,A -85,B 0,C 180,E1 -5745.451,E2 -5745.451} C_VEL
LIN {X 0,Y 502.96,Z 333.616,A -85,B 0,C 180,E1 -5745.588,E2 -5745.588} C_VEL
LIN {X 0,Y 502.825,Z 332.876,A -85,B 0,C 180,E1 -5745.79,E2 -5745.79} C_VEL
LIN {X 0,Y 502.877,Z 332.845,A -85,B 0,C 180,E1 -5748.717,E2 -5748.717} C_VEL
LIN {X 0,Y 502.891,Z 332.842,A -85,B 0,C 180,E1 -5751.967,E2 -5751.967} C_VEL
LIN {X 0,Y 502.921,Z 332.836,A -85,B 0,C 180,E1 -5754.386,E2 -5754.386} C_VEL
LIN {X 0,Y 503.011,Z 332.829,A -85,B 0,C 180,E1 -5757.598,E2 -5757.598} C_VEL
LIN {X 0,Y 503.012,Z 332.825,A -85,B 0,C 180,E1 -5760,E2 -5760} C_VEL
LIN {X 0,Y 503.01,Z 332.824,A -85,B 0,C 180,E1 -5762.402,E2 -5762.402} C_VEL
LIN {X 0,Y 502.92,Z 332.839,A -85,B 0,C 180,E1 -5765.614,E2 -5765.614} C_VEL
LIN {X 0,Y 502.869,Z 332.841,A -85,B 0,C 180,E1 -5768.034,E2 -5768.034} C_VEL
LIN {X 0,Y 502.865,Z 332.848,A -85,B 0,C 180,E1 -5771.284,E2 -5771.284} C_VEL
LIN {X 0,Y 502.833,Z 332.848,A -85,B 0,C 180,E1 -5774.571,E2 -5774.571} C_VEL
LIN {X 0,Y 502.811,Z 332.847,A -85,B 0,C 180,E1 -5777.909,E2 -5777.909} C_VEL
LIN {X 0,Y 502.819,Z 332.849,A -85,B 0,C 180,E1 -5780.537,E2 -5780.537} C_VEL
LIN {X 0,Y 502.777,Z 332.858,A -85,B 0,C 180,E1 -5783.041,E2 -5783.041} C_VEL
LIN {X 0,Y 502.817,Z 332.848,A -85,B 0,C 180,E1 -5785.677,E2 -5785.677} C_VEL
LIN {X 0,Y 502.828,Z 332.849,A -85,B 0,C 180,E1 -5788.374,E2 -5788.374} C_VEL
LIN {X 0,Y 502.783,Z 332.854,A -85,B 0,C 180,E1 -5791.499,E2 -5791.499} C_VEL
LIN {X 0,Y 502.781,Z 332.853,A -85,B 0,C 180,E1 -5793.996,E2 -5793.996} C_VEL
LIN {X 0,Y 502.769,Z 332.859,A -85,B 0,C 180,E1 -5797.178,E2 -5797.178} C_VEL
LIN {X 0,Y 502.764,Z 332.856,A -85,B 0,C 180,E1 -5800.018,E2 -5800.018} C_VEL
LIN {X 0,Y 502.744,Z 332.861,A -85,B 0,C 180,E1 -5803.235,E2 -5803.235} C_VEL
LIN {X 0,Y 502.773,Z 332.856,A -85,B 0,C 180,E1 -5805.661,E2 -5805.661} C_VEL
LIN {X 0,Y 502.767,Z 332.86,A -85,B 0,C 180,E1 -5808.93,E2 -5808.93} C_VEL
LIN {X 0,Y 502.798,Z 332.954,A -85,B 0,C 180,E1 -5811.514,E2 -5811.514} C_VEL
LIN {X 0,Y 504.29,Z 340.653,A -85,B 0,C 180,E1 -5813.591,E2 -5813.591} C_VEL
LIN {X 0,Y 504.389,Z 345.028,A -85,B 0,C 180,E1 -5814.674,E2 -5814.674} C_VEL
LIN {X 0,Y 503.825,Z 359.263,A -85,B 0,C 180,E1 -5817.991,E2 -5817.991} C_VEL
LIN {X 0,Y 503.605,Z 371.695,A -85,B 0,C 180,E1 -5820.763,E2 -5820.763} C_VEL
LIN {X 0,Y 503.378,Z 386.35,A -85,B 0,C 180,E1 -5823.91,E2 -5823.91} C_VEL
LIN {X 0,Y 503.127,Z 402.2,A -85,B 0,C 180,E1 -5827.21,E2 -5827.21} C_VEL
LIN {X 0,Y 502.95,Z 416.836,A -85,B 0,C 180,E1 -5830.193,E2 -5830.193} C_VEL
LIN {X 0,Y 502.79,Z 430.44,A -85,B 0,C 180,E1 -5832.931,E2 -5832.931} C_VEL
LIN {X 0,Y 502.615,Z 444.139,A -85,B 0,C 180,E1 -5835.63,E2 -5835.63} C_VEL
LIN {X 0,Y 502.765,Z 446.11,A -85,B 0,C 180,E1 -5835.711,E2 -5835.711} C_VEL
LIN {X 0,Y 503.782,Z 456.792,A -85,B 0,C 180,E1 -5835.973,E2 -5835.973} C_VEL
LIN {X 0,Y 504.417,Z 462.115,A -85,B 0,C 180,E1 -5836.145,E2 -5836.145} C_VEL
LIN {X 0,Y 504.09,Z 475.21,A -85,B 0,C 180,E1 -5836.649,E2 -5836.649} C_VEL
LIN {X 0,Y 503.781,Z 487.499,A -85,B 0,C 180,E1 -5837.291,E2 -5837.291} C_VEL
LIN {X 0,Y 503.506,Z 498.399,A -85,B 0,C 180,E1 -5838.017,E2 -5838.017} C_VEL
LIN {X 0,Y 503.135,Z 509.326,A -85,B 0,C 180,E1 -5838.927,E2 -5838.927} C_VEL
LIN {X 0,Y 502.803,Z 519.193,A -85,B 0,C 180,E1 -5839.938,E2 -5839.938} C_VEL
LIN {X 0,Y 502.63,Z 527.332,A -85,B 0,C 180,E1 -5840.95,E2 -5840.95} C_VEL
LIN {X 0,Y 502.454,Z 535.327,A -85,B 0,C 180,E1 -5842.162,E2 -5842.162} C_VEL
LIN {X 0,Y 502.323,Z 542.654,A -85,B 0,C 180,E1 -5843.574,E2 -5843.574} C_VEL
LIN {X 0,Y 502.27,Z 547.553,A -85,B 0,C 180,E1 -5844.782,E2 -5844.782} C_VEL
LIN {X 0,Y 502.294,Z 551.311,A -85,B 0,C 180,E1 -5845.988,E2 -5845.988} C_VEL
LIN {X 0,Y 502.203,Z 553.237,A -85,B 0,C 180,E1 -5846.791,E2 -5846.791} C_VEL
LIN {X 0,Y 502.183,Z 554.694,A -85,B 0,C 180,E1 -5847.594,E2 -5847.594} C_VEL
LIN {X 0,Y 502.147,Z 556.37,A -85,B 0,C 180,E1 -5849.198,E2 -5849.198} C_VEL
LIN {X 0,Y 502.138,Z 556.603,A -85,B 0,C 180,E1 -5850,E2 -5850} C_VEL
LIN {X 0,Y 502.147,Z 556.392,A -85,B 0,C 180,E1 -5850.802,E2 -5850.802} C_VEL
LIN {X 0,Y 502.175,Z 554.771,A -85,B 0,C 180,E1 -5852.406,E2 -5852.406} C_VEL
LIN {X 0,Y 502.193,Z 553.338,A -85,B 0,C 180,E1 -5853.209,E2 -5853.209} C_VEL
LIN {X 0,Y 502.216,Z 550.337,A -85,B 0,C 180,E1 -5854.414,E2 -5854.414} C_VEL
LIN {X 0,Y 502.282,Z 546.27,A -85,B 0,C 180,E1 -5855.621,E2 -5855.621} C_VEL
LIN {X 0,Y 502.336,Z 540.098,A -85,B 0,C 180,E1 -5857.011,E2 -5857.011} C_VEL
LIN {X 0,Y 502.496,Z 533.175,A -85,B 0,C 180,E1 -5858.242,E2 -5858.242} C_VEL
LIN {X 0,Y 502.682,Z 524.711,A -85,B 0,C 180,E1 -5859.455,E2 -5859.455} C_VEL
LIN {X 0,Y 502.954,Z 516.021,A -85,B 0,C 180,E1 -5860.466,E2 -5860.466} C_VEL
LIN {X 0,Y 503.274,Z 505.366,A -85,B 0,C 180,E1 -5861.478,E2 -5861.478} C_VEL
LIN {X 0,Y 503.612,Z 494.9,A -85,B 0,C 180,E1 -5862.284,E2 -5862.284} C_VEL
LIN {X 0,Y 503.93,Z 483.255,A -85,B 0,C 180,E1 -5862.996,E2 -5862.996} C_VEL
LIN {X 0,Y 504.337,Z 470.151,A -85,B 0,C 180,E1 -5863.6,E2 -5863.6} C_VEL
LIN {X 0,Y 504.28,Z 459.649,A -85,B 0,C 180,E1 -5863.962,E2 -5863.962} C_VEL
LIN {X 0,Y 502.906,Z 448.718,A -85,B 0,C 180,E1 -5864.259,E2 -5864.259} C_VEL
LIN {X 0,Y 502.615,Z 445.234,A -85,B 0,C 180,E1 -5864.37,E2 -5864.37} C_VEL
LIN {X 0,Y 502.77,Z 433.891,A -85,B 0,C 180,E1 -5866.652,E2 -5866.652} C_VEL
LIN {X 0,Y 503.012,Z 419.692,A -85,B 0,C 180,E1 -5869.592,E2 -5869.592} C_VEL
LIN {X 0,Y 503.304,Z 405.884,A -85,B 0,C 180,E1 -5872.495,E2 -5872.495} C_VEL
LIN {X 0,Y 503.628,Z 391.294,A -85,B 0,C 180,E1 -5875.632,E2 -5875.632} C_VEL
LIN {X 0,Y 503.998,Z 376.842,A -85,B 0,C 180,E1 -5878.82,E2 -5878.82} C_VEL
LIN {X 0,Y 504.351,Z 363.756,A -85,B 0,C 180,E1 -5881.786,E2 -5881.786} C_VEL
LIN {X 0,Y 505.056,Z 348.834,A -85,B 0,C 180,E1 -5885.273,E2 -5885.273} C_VEL
LIN {X 0,Y 504.993,Z 344.078,A -85,B 0,C 180,E1 -5886.435,E2 -5886.435} C_VEL
LIN {X 0,Y 503.129,Z 334.521,A -85,B 0,C 180,E1 -5888.945,E2 -5888.945} C_VEL
LIN {X 0,Y 502.784,Z 332.932,A -85,B 0,C 180,E1 -5889.429,E2 -5889.429} C_VEL
LIN {X 0,Y 502.766,Z 332.858,A -85,B 0,C 180,E1 -5892.194,E2 -5892.194} C_VEL
LIN {X 0,Y 502.78,Z 332.86,A -85,B 0,C 180,E1 -5895.469,E2 -5895.469} C_VEL
LIN {X 0,Y 502.764,Z 332.857,A -85,B 0,C 180,E1 -5898.928,E2 -5898.928} C_VEL
LIN {X 0,Y 502.784,Z 332.852,A -85,B 0,C 180,E1 -5902.045,E2 -5902.045} C_VEL
LIN {X 0,Y 502.787,Z 332.856,A -85,B 0,C 180,E1 -5905.033,E2 -5905.033} C_VEL
LIN {X 0,Y 502.773,Z 332.853,A -85,B 0,C 180,E1 -5907.915,E2 -5907.915} C_VEL
LIN {X 0,Y 502.814,Z 332.849,A -85,B 0,C 180,E1 -5910.711,E2 -5910.711} C_VEL
LIN {X 0,Y 502.854,Z 332.847,A -85,B 0,C 180,E1 -5913.439,E2 -5913.439} C_VEL
LIN {X 0,Y 502.763,Z 332.854,A -85,B 0,C 180,E1 -5916.085,E2 -5916.085} C_VEL
LIN {X 0,Y 502.772,Z 332.856,A -85,B 0,C 180,E1 -5918.688,E2 -5918.688} C_VEL
LIN {X 0,Y 502.815,Z 332.853,A -85,B 0,C 180,E1 -5921.248,E2 -5921.248} C_VEL
LIN {X 0,Y 502.838,Z 332.847,A -85,B 0,C 180,E1 -5924.6,E2 -5924.6} C_VEL
LIN {X 0,Y 502.865,Z 332.841,A -85,B 0,C 180,E1 -5928.039,E2 -5928.039} C_VEL
LIN {X 0,Y 502.854,Z 332.848,A -85,B 0,C 180,E1 -5931.156,E2 -5931.156} C_VEL
LIN {X 0,Y 502.893,Z 332.838,A -85,B 0,C 180,E1 -5933.581,E2 -5933.581} C_VEL
LIN {X 0,Y 502.887,Z 332.846,A -85,B 0,C 180,E1 -5936.795,E2 -5936.795} C_VEL
LIN {X 0,Y 503.023,Z 332.825,A -85,B 0,C 180,E1 -5939.199,E2 -5939.199} C_VEL
LIN {X 0,Y 502.887,Z 332.838,A -85,B 0,C 180,E1 -5941.602,E2 -5941.602} C_VEL
LIN {X 0,Y 502.886,Z 332.841,A -85,B 0,C 180,E1 -5943.205,E2 -5943.205} C_VEL
LIN {X 0,Y 502.894,Z 332.842,A -85,B 0,C 180,E1 -5946.419,E2 -5946.419} C_VEL
LIN {X 0,Y 502.863,Z 332.848,A -85,B 0,C 180,E1 -5948.843,E2 -5948.843} C_VEL
LIN {X 0,Y 502.836,Z 332.847,A -85,B 0,C 180,E1 -5952.102,E2 -5952.102} C_VEL
LIN {X 0,Y 502.838,Z 332.845,A -85,B 0,C 180,E1 -5955.4,E2 -5955.4} C_VEL
LIN {X 0,Y 502.836,Z 332.848,A -85,B 0,C 180,E1 -5958.123,E2 -5958.123} C_VEL
LIN {X 0,Y 502.787,Z 332.851,A -85,B 0,C 180,E1 -5961.311,E2 -5961.311} C_VEL
LIN {X 0,Y 502.793,Z 332.852,A -85,B 0,C 180,E1 -5963.914,E2 -5963.914} C_VEL
LIN {X 0,Y 502.855,Z 332.849,A -85,B 0,C 180,E1 -5966.567,E2 -5966.567} C_VEL
LIN {X 0,Y 502.831,Z 332.845,A -85,B 0,C 180,E1 -5969.287,E2 -5969.287} C_VEL
LIN {X 0,Y 502.777,Z 332.857,A -85,B 0,C 180,E1 -5972.085,E2 -5972.085} C_VEL
LIN {X 0,Y 502.8,Z 332.85,A -85,B 0,C 180,E1 -5974.966,E2 -5974.966} C_VEL
LIN {X 0,Y 502.787,Z 332.855,A -85,B 0,C 180,E1 -5977.955,E2 -5977.955} C_VEL
LIN {X 0,Y 502.821,Z 332.847,A -85,B 0,C 180,E1 -5981.066,E2 -5981.066} C_VEL
LIN {X 0,Y 502.796,Z 332.853,A -85,B 0,C 180,E1 -5984.533,E2 -5984.533} C_VEL
LIN {X 0,Y 502.826,Z 332.851,A -85,B 0,C 180,E1 -5987.865,E2 -5987.865} C_VEL
LIN {X 0,Y 502.798,Z 332.849,A -85,B 0,C 180,E1 -5991.025,E2 -5991.025} C_VEL
LIN {X 0,Y 502.782,Z 332.858,A -85,B 0,C 180,E1 -5994.168,E2 -5994.168} C_VEL
LIN {X 0,Y 502.805,Z 332.849,A -85,B 0,C 180,E1 -5997.243,E2 -5997.243} C_VEL
LIN {X 0,Y 502.107,Z 332.943,A -85,B 0,C 180,E1 -5997.912,E2 -5997.912} C_VEL
LIN {X 0,Y 499.25,Z 333.296,A -85,B 0,C 180,E1 -5998.998,E2 -5998.998} C_VEL
LIN {X 0,Y 496.86,Z 333.597,A -85,B 0,C 180,E1 -5999.873,E2 -5999.873} C_VEL
LIN {X 0,Y 495.843,Z 333.717,A -85,B 0,C 180,E1 -6000.548,E2 -6000.548} C_VEL
LIN {X 0,Y 495.764,Z 333.726,A -85,B 0,C 180,E1 -6000.777,E2 -6000.777} C_VEL
LIN {X 0,Y 495.801,Z 333.73,A -85,B 0,C 180,E1 -6003.933,E2 -6003.933} C_VEL
LIN {X 0,Y 495.766,Z 333.726,A -85,B 0,C 180,E1 -6007.138,E2 -6007.138} C_VEL
LIN {X 0,Y 495.779,Z 333.728,A -85,B 0,C 180,E1 -6010.111,E2 -6010.111} C_VEL
LIN {X 0,Y 495.788,Z 333.723,A -85,B 0,C 180,E1 -6012.682,E2 -6012.682} C_VEL
LIN {X 0,Y 495.792,Z 333.724,A -85,B 0,C 180,E1 -6015.218,E2 -6015.218} C_VEL
LIN {X 0,Y 495.854,Z 333.714,A -85,B 0,C 180,E1 -6018.555,E2 -6018.555} C_VEL
LIN {X 0,Y 495.876,Z 333.717,A -85,B 0,C 180,E1 -6021.852,E2 -6021.852} C_VEL
LIN {X 0,Y 495.902,Z 333.709,A -85,B 0,C 180,E1 -6024.307,E2 -6024.307} C_VEL
LIN {X 0,Y 495.997,Z 333.705,A -85,B 0,C 180,E1 -6027.564,E2 -6027.564} C_VEL
LIN {X 0,Y 496.002,Z 333.698,A -85,B 0,C 180,E1 -6030,E2 -6030} C_VEL
LIN {X 0,Y 495.997,Z 333.696,A -85,B 0,C 180,E1 -6032.436,E2 -6032.436} C_VEL
LIN {X 0,Y 495.893,Z 333.715,A -85,B 0,C 180,E1 -6035.693,E2 -6035.693} C_VEL
LIN {X 0,Y 495.876,Z 333.712,A -85,B 0,C 180,E1 -6038.148,E2 -6038.148} C_VEL
LIN {X 0,Y 495.854,Z 333.722,A -85,B 0,C 180,E1 -6041.445,E2 -6041.445} C_VEL
LIN {X 0,Y 495.793,Z 333.724,A -85,B 0,C 180,E1 -6044.782,E2 -6044.782} C_VEL
LIN {X 0,Y 495.791,Z 333.731,A -85,B 0,C 180,E1 -6047.318,E2 -6047.318} C_VEL
LIN {X 0,Y 495.78,Z 333.725,A -85,B 0,C 180,E1 -6049.889,E2 -6049.889} C_VEL
LIN {X 0,Y 495.766,Z 333.729,A -85,B 0,C 180,E1 -6052.862,E2 -6052.862} C_VEL
LIN {X 0,Y 495.8,Z 333.721,A -85,B 0,C 180,E1 -6056.067,E2 -6056.067} C_VEL
LIN {X 0,Y 495.772,Z 333.729,A -85,B 0,C 180,E1 -6058.814,E2 -6058.814} C_VEL
LIN {X 0,Y 495.758,Z 333.728,A -85,B 0,C 180,E1 -6061.725,E2 -6061.725} C_VEL
LIN {X 0,Y 495.775,Z 333.728,A -85,B 0,C 180,E1 -6064.695,E2 -6064.695} C_VEL
LIN {X 0,Y 495.733,Z 333.731,A -85,B 0,C 180,E1 -6067.56,E2 -6067.56} C_VEL
LIN {X 0,Y 495.791,Z 333.724,A -85,B 0,C 180,E1 -6070.051,E2 -6070.051} C_VEL
LIN {X 0,Y 495.76,Z 333.734,A -85,B 0,C 180,E1 -6072.878,E2 -6072.878} C_VEL
LIN {X 0,Y 495.732,Z 333.733,A -85,B 0,C 180,E1 -6075.999,E2 -6075.999} C_VEL
LIN {X 0,Y 495.844,Z 333.956,A -85,B 0,C 180,E1 -6078.273,E2 -6078.273} C_VEL
LIN {X 0,Y 496.195,Z 335.315,A -85,B 0,C 180,E1 -6078.424,E2 -6078.424} C_VEL
LIN {X 0,Y 497.661,Z 340.897,A -85,B 0,C 180,E1 -6078.753,E2 -6078.753} C_VEL
LIN {X 0,Y 497.456,Z 352.767,A -85,B 0,C 180,E1 -6079.467,E2 -6079.467} C_VEL
LIN {X 0,Y 497.101,Z 362.986,A -85,B 0,C 180,E1 -6080.239,E2 -6080.239} C_VEL
LIN {X 0,Y 496.815,Z 372.058,A -85,B 0,C 180,E1 -6081.079,E2 -6081.079} C_VEL
LIN {X 0,Y 496.518,Z 380.694,A -85,B 0,C 180,E1 -6082.047,E2 -6082.047} C_VEL
LIN {X 0,Y 496.179,Z 389.355,A -85,B 0,C 180,E1 -6083.242,E2 -6083.242} C_VEL
LIN {X 0,Y 495.896,Z 396.57,A -85,B 0,C 180,E1 -6084.474,E2 -6084.474} C_VEL
LIN {X 0,Y 495.699,Z 402.308,A -85,B 0,C 180,E1 -6085.697,E2 -6085.697} C_VEL
LIN {X 0,Y 495.542,Z 406.419,A -85,B 0,C 180,E1 -6086.798,E2 -6086.798} C_VEL
LIN {X 0,Y 495.478,Z 410.72,A -85,B 0,C 180,E1 -6088.344,E2 -6088.344} C_VEL
LIN {X 0,Y 495.361,Z 413.551,A -85,B 0,C 180,E1 -6089.931,E2 -6089.931} C_VEL
LIN {X 0,Y 495.309,Z 414.868,A -85,B 0,C 180,E1 -6091.607,E2 -6091.607} C_VEL
LIN {X 0,Y 495.324,Z 414.506,A -85,B 0,C 180,E1 -6093.363,E2 -6093.363} C_VEL
LIN {X 0,Y 495.412,Z 412.793,A -85,B 0,C 180,E1 -6094.812,E2 -6094.812} C_VEL
LIN {X 0,Y 495.548,Z 410.055,A -85,B 0,C 180,E1 -6096.159,E2 -6096.159} C_VEL
LIN {X 0,Y 495.685,Z 406.172,A -85,B 0,C 180,E1 -6097.492,E2 -6097.492} C_VEL
LIN {X 0,Y 495.873,Z 401.044,A -85,B 0,C 180,E1 -6098.813,E2 -6098.813} C_VEL
LIN {X 0,Y 496.115,Z 394.47,A -85,B 0,C 180,E1 -6100.124,E2 -6100.124} C_VEL
LIN {X 0,Y 496.414,Z 386.914,A -85,B 0,C 180,E1 -6101.324,E2 -6101.324} C_VEL
LIN {X 0,Y 496.764,Z 377.71,A -85,B 0,C 180,E1 -6102.504,E2 -6102.504} C_VEL
LIN {X 0,Y 497.133,Z 367.155,A -85,B 0,C 180,E1 -6103.576,E2 -6103.576} C_VEL
LIN {X 0,Y 497.51,Z 356.651,A -85,B 0,C 180,E1 -6104.431,E2 -6104.431} C_VEL
LIN {X 0,Y 497.83,Z 345.053,A -85,B 0,C 180,E1 -6105.175,E2 -6105.175} C_VEL
LIN {X 0,Y 497.803,Z 341.296,A -85,B 0,C 180,E1 -6105.383,E2 -6105.383} C_VEL
LIN {X 0,Y 495.91,Z 334.462,A -85,B 0,C 180,E1 -6105.797,E2 -6105.797} C_VEL
LIN {X 0,Y 495.799,Z 333.749,A -85,B 0,C 180,E1 -6106.003,E2 -6106.003} C_VEL
LIN {X 0,Y 495.859,Z 333.719,A -85,B 0,C 180,E1 -6108.555,E2 -6108.555} C_VEL
LIN {X 0,Y 495.862,Z 333.719,A -85,B 0,C 180,E1 -6111.852,E2 -6111.852} C_VEL
LIN {X 0,Y 495.877,Z 333.714,A -85,B 0,C 180,E1 -6114.306,E2 -6114.306} C_VEL
LIN {X 0,Y 495.98,Z 333.706,A -85,B 0,C 180,E1 -6117.564,E2 -6117.564} C_VEL
LIN {X 0,Y 495.983,Z 333.701,A -85,B 0,C 180,E1 -6120,E2 -6120} C_VEL
LIN {X 0,Y 495.979,Z 333.7,A -85,B 0,C 180,E1 -6122.436,E2 -6122.436} C_VEL
LIN {X 0,Y 495.876,Z 333.715,A -85,B 0,C 180,E1 -6125.694,E2 -6125.694} C_VEL
LIN {X 0,Y 495.825,Z 333.718,A -85,B 0,C 180,E1 -6128.149,E2 -6128.149} C_VEL
LIN {X 0,Y 495.84,Z 333.721,A -85,B 0,C 180,E1 -6131.446,E2 -6131.446} C_VEL
LIN {X 0,Y 495.778,Z 333.729,A -85,B 0,C 180,E1 -6134.783,E2 -6134.783} C_VEL
LIN {X 0,Y 495.753,Z 333.73,A -85,B 0,C 180,E1 -6137.32,E2 -6137.32} C_VEL
LIN {X 0,Y 495.76,Z 333.727,A -85,B 0,C 180,E1 -6139.891,E2 -6139.891} C_VEL
LIN {X 0,Y 495.748,Z 333.736,A -85,B 0,C 180,E1 -6142.861,E2 -6142.861} C_VEL
LIN {X 0,Y 495.774,Z 333.725,A -85,B 0,C 180,E1 -6146.069,E2 -6146.069} C_VEL
LIN {X 0,Y 495.761,Z 333.733,A -85,B 0,C 180,E1 -6148.816,E2 -6148.816} C_VEL
LIN {X 0,Y 495.745,Z 333.73,A -85,B 0,C 180,E1 -6151.726,E2 -6151.726} C_VEL
LIN {X 0,Y 495.754,Z 333.735,A -85,B 0,C 180,E1 -6154.693,E2 -6154.693} C_VEL
LIN {X 0,Y 495.72,Z 333.734,A -85,B 0,C 180,E1 -6157.563,E2 -6157.563} C_VEL
LIN {X 0,Y 495.736,Z 333.732,A -85,B 0,C 180,E1 -6160.046,E2 -6160.046} C_VEL
LIN {X 0,Y 495.698,Z 333.742,A -85,B 0,C 180,E1 -6162.886,E2 -6162.886} C_VEL
LIN {X 0,Y 495.718,Z 333.736,A -85,B 0,C 180,E1 -6165.999,E2 -6165.999} C_VEL
LIN {X 0,Y 495.726,Z 333.735,A -85,B 0,C 180,E1 -6169.297,E2 -6169.297} C_VEL
LIN {X 0,Y 495.808,Z 333.962,A -85,B 0,C 180,E1 -6171.306,E2 -6171.306} C_VEL
LIN {X 0,Y 497.415,Z 342.508,A -85,B 0,C 180,E1 -6173.645,E2 -6173.645} C_VEL
LIN {X 0,Y 497.378,Z 348.144,A -85,B 0,C 180,E1 -6175.04,E2 -6175.04} C_VEL
LIN {X 0,Y 496.763,Z 363.574,A -85,B 0,C 180,E1 -6178.674,E2 -6178.674} C_VEL
LIN {X 0,Y 496.519,Z 375.478,A -85,B 0,C 180,E1 -6181.352,E2 -6181.352} C_VEL
LIN {X 0,Y 496.276,Z 389.546,A -85,B 0,C 180,E1 -6184.411,E2 -6184.411} C_VEL
LIN {X 0,Y 496.013,Z 405.259,A -85,B 0,C 180,E1 -6187.728,E2 -6187.728} C_VEL
LIN {X 0,Y 495.837,Z 419.926,A -85,B 0,C 180,E1 -6190.759,E2 -6190.759} C_VEL
LIN {X 0,Y 495.645,Z 434.51,A -85,B 0,C 180,E1 -6193.738,E2 -6193.738} C_VEL
LIN {X 0,Y 495.536,Z 442.972,A -85,B 0,C 180,E1 -6195.42,E2 -6195.42} C_VEL
LIN {X 0,Y 495.642,Z 444.79,A -85,B 0,C 180,E1 -6195.502,E2 -6195.502} C_VEL
LIN {X 0,Y 496.807,Z 457.266,A -85,B 0,C 180,E1 -6195.824,E2 -6195.824} C_VEL
LIN {X 0,Y 497.423,Z 463.81,A -85,B 0,C 180,E1 -6196.05,E2 -6196.05} C_VEL
LIN {X 0,Y 497.052,Z 477.256,A -85,B 0,C 180,E1 -6196.613,E2 -6196.613} C_VEL
LIN {X 0,Y 496.722,Z 488.705,A -85,B 0,C 180,E1 -6197.259,E2 -6197.259} C_VEL
LIN {X 0,Y 496.43,Z 499.817,A -85,B 0,C 180,E1 -6198.051,E2 -6198.051} C_VEL
LIN {X 0,Y 496.061,Z 510.322,A -85,B 0,C 180,E1 -6198.974,E2 -6198.974} C_VEL
LIN {X 0,Y 495.715,Z 519.83,A -85,B 0,C 180,E1 -6199.999,E2 -6199.999} C_VEL
LIN {X 0,Y 495.479,Z 529.053,A -85,B 0,C 180,E1 -6201.23,E2 -6201.23} C_VEL
LIN {X 0,Y 495.334,Z 536.521,A -85,B 0,C 180,E1 -6202.459,E2 -6202.459} C_VEL
LIN {X 0,Y 495.252,Z 541.575,A -85,B 0,C 180,E1 -6203.482,E2 -6203.482} C_VEL
LIN {X 0,Y 495.222,Z 546.497,A -85,B 0,C 180,E1 -6204.707,E2 -6204.707} C_VEL
LIN {X 0,Y 495.249,Z 550.273,A -85,B 0,C 180,E1 -6205.931,E2 -6205.931} C_VEL
LIN {X 0,Y 495.163,Z 552.213,A -85,B 0,C 180,E1 -6206.745,E2 -6206.745} C_VEL
LIN {X 0,Y 495.144,Z 553.678,A -85,B 0,C 180,E1 -6207.56,E2 -6207.56} C_VEL
LIN {X 0,Y 495.136,Z 555.37,A -85,B 0,C 180,E1 -6209.187,E2 -6209.187} C_VEL
LIN {X 0,Y 495.125,Z 555.612,A -85,B 0,C 180,E1 -6210,E2 -6210} C_VEL
LIN {X 0,Y 495.136,Z 555.405,A -85,B 0,C 180,E1 -6210.813,E2 -6210.813} C_VEL
LIN {X 0,Y 495.132,Z 553.786,A -85,B 0,C 180,E1 -6212.44,E2 -6212.44} C_VEL
LIN {X 0,Y 495.149,Z 552.356,A -85,B 0,C 180,E1 -6213.255,E2 -6213.255} C_VEL
LIN {X 0,Y 495.155,Z 549.355,A -85,B 0,C 180,E1 -6214.477,E2 -6214.477} C_VEL
LIN {X 0,Y 495.262,Z 544.074,A -85,B 0,C 180,E1 -6216.005,E2 -6216.005} C_VEL
LIN {X 0,Y 495.276,Z 537.987,A -85,B 0,C 180,E1 -6217.337,E2 -6217.337} C_VEL
LIN {X 0,Y 495.45,Z 530.918,A -85,B 0,C 180,E1 -6218.565,E2 -6218.565} C_VEL
LIN {X 0,Y 495.653,Z 522.075,A -85,B 0,C 180,E1 -6219.796,E2 -6219.796} C_VEL
LIN {X 0,Y 496.059,Z 512.095,A -85,B 0,C 180,E1 -6220.923,E2 -6220.923} C_VEL
LIN {X 0,Y 496.403,Z 501.948,A -85,B 0,C 180,E1 -6221.846,E2 -6221.846} C_VEL
LIN {X 0,Y 496.706,Z 490.704,A -85,B 0,C 180,E1 -6222.672,E2 -6222.672} C_VEL
LIN {X 0,Y 497.117,Z 478.351,A -85,B 0,C 180,E1 -6223.385,E2 -6223.385} C_VEL
LIN {X 0,Y 497.435,Z 465.74,A -85,B 0,C 180,E1 -6223.923,E2 -6223.923} C_VEL
LIN {X 0,Y 497.299,Z 460.343,A -85,B 0,C 180,E1 -6224.11,E2 -6224.11} C_VEL
LIN {X 0,Y 495.971,Z 449.013,A -85,B 0,C 180,E1 -6224.436,E2 -6224.436} C_VEL
LIN {X 0,Y 495.536,Z 444.33,A -85,B 0,C 180,E1 -6224.58,E2 -6224.58} C_VEL
LIN {X 0,Y 495.687,Z 434.046,A -85,B 0,C 180,E1 -6226.685,E2 -6226.685} C_VEL
LIN {X 0,Y 495.954,Z 419.923,A -85,B 0,C 180,E1 -6229.666,E2 -6229.666} C_VEL
LIN {X 0,Y 496.275,Z 405.578,A -85,B 0,C 180,E1 -6232.741,E2 -6232.741} C_VEL
LIN {X 0,Y 496.628,Z 390.588,A -85,B 0,C 180,E1 -6236.02,E2 -6236.02} C_VEL
LIN {X 0,Y 497.047,Z 376.453,A -85,B 0,C 180,E1 -6239.196,E2 -6239.196} C_VEL
LIN {X 0,Y 497.425,Z 364.161,A -85,B 0,C 180,E1 -6242.035,E2 -6242.035} C_VEL
LIN {X 0,Y 498.122,Z 350.223,A -85,B 0,C 180,E1 -6245.342,E2 -6245.342} C_VEL
LIN {X 0,Y 498.095,Z 345.719,A -85,B 0,C 180,E1 -6246.461,E2 -6246.461} C_VEL
LIN {X 0,Y 496.096,Z 335.499,A -85,B 0,C 180,E1 -6249.184,E2 -6249.184} C_VEL
LIN {X 0,Y 495.732,Z 333.819,A -85,B 0,C 180,E1 -6249.69,E2 -6249.69} C_VEL
LIN {X 0,Y 495.699,Z 333.74,A -85,B 0,C 180,E1 -6252.885,E2 -6252.885} C_VEL
LIN {X 0,Y 495.717,Z 333.735,A -85,B 0,C 180,E1 -6255.997,E2 -6255.997} C_VEL
LIN {X 0,Y 495.724,Z 333.738,A -85,B 0,C 180,E1 -6259.296,E2 -6259.296} C_VEL
LIN {X 0,Y 495.738,Z 333.737,A -85,B 0,C 180,E1 -6261.407,E2 -6261.407} C_VEL
LIN {X 0,Y 495.739,Z 333.729,A -85,B 0,C 180,E1 -6264.461,E2 -6264.461} C_VEL
LIN {X 0,Y 495.757,Z 333.733,A -85,B 0,C 180,E1 -6267.405,E2 -6267.405} C_VEL
LIN {X 0,Y 495.757,Z 333.726,A -85,B 0,C 180,E1 -6270.253,E2 -6270.253} C_VEL
LIN {X 0,Y 495.814,Z 333.727,A -85,B 0,C 180,E1 -6273.25,E2 -6273.25} C_VEL
LIN {X 0,Y 495.731,Z 333.732,A -85,B 0,C 180,E1 -6276.612,E2 -6276.612} C_VEL
LIN {X 0,Y 495.769,Z 333.73,A -85,B 0,C 180,E1 -6279.324,E2 -6279.324} C_VEL
LIN {X 0,Y 495.77,Z 333.725,A -85,B 0,C 180,E1 -6281.828,E2 -6281.828} C_VEL
LIN {X 0,Y 495.813,Z 333.722,A -85,B 0,C 180,E1 -6284.548,E2 -6284.548} C_VEL
LIN {X 0,Y 495.817,Z 333.719,A -85,B 0,C 180,E1 -6287.965,E2 -6287.965} C_VEL
LIN {X 0,Y 495.825,Z 333.725,A -85,B 0,C 180,E1 -6291.03,E2 -6291.03} C_VEL
LIN {X 0,Y 495.848,Z 333.717,A -85,B 0,C 180,E1 -6293.489,E2 -6293.489} C_VEL
LIN {X 0,Y 495.831,Z 333.725,A -85,B 0,C 180,E1 -6296.75,E2 -6296.75} C_VEL
LIN {X 0,Y 495.994,Z 333.7,A -85,B 0,C 180,E1 -6299.188,E2 -6299.188} C_VEL
LIN {X 0,Y 495.857,Z 333.714,A -85,B 0,C 180,E1 -6301.624,E2 -6301.624} C_VEL
LIN {X 0,Y 495.829,Z 333.72,A -85,B 0,C 180,E1 -6303.25,E2 -6303.25} C_VEL
LIN {X 0,Y 495.848,Z 333.721,A -85,B 0,C 180,E1 -6306.511,E2 -6306.511} C_VEL
LIN {X 0,Y 495.832,Z 333.722,A -85,B 0,C 180,E1 -6308.97,E2 -6308.97} C_VEL
LIN {X 0,Y 495.818,Z 333.72,A -85,B 0,C 180,E1 -6312.035,E2 -6312.035} C_VEL
LIN {X 0,Y 495.813,Z 333.719,A -85,B 0,C 180,E1 -6315.452,E2 -6315.452} C_VEL
LIN {X 0,Y 495.797,Z 333.726,A -85,B 0,C 180,E1 -6318.248,E2 -6318.248} C_VEL
LIN {X 0,Y 495.767,Z 333.73,A -85,B 0,C 180,E1 -6320.757,E2 -6320.757} C_VEL
LIN {X 0,Y 495.752,Z 333.727,A -85,B 0,C 180,E1 -6323.387,E2 -6323.387} C_VEL
LIN {X 0,Y 495.782,Z 333.727,A -85,B 0,C 180,E1 -6326.068,E2 -6326.068} C_VEL
LIN {X 0,Y 495.772,Z 333.728,A -85,B 0,C 180,E1 -6328.815,E2 -6328.815} C_VEL
LIN {X 0,Y 495.748,Z 333.729,A -85,B 0,C 180,E1 -6331.726,E2 -6331.726} C_VEL
LIN {X 0,Y 495.767,Z 333.729,A -85,B 0,C 180,E1 -6334.696,E2 -6334.696} C_VEL
LIN {X 0,Y 495.724,Z 333.731,A -85,B 0,C 180,E1 -6337.562,E2 -6337.562} C_VEL
LIN {X 0,Y 495.773,Z 333.727,A -85,B 0,C 180,E1 -6340.699,E2 -6340.699} C_VEL
LIN {X 0,Y 495.729,Z 333.736,A -85,B 0,C 180,E1 -6344.002,E2 -6344.002} C_VEL
LIN {X 0,Y 495.729,Z 333.73,A -85,B 0,C 180,E1 -6347.119,E2 -6347.119} C_VEL
LIN {X 0,Y 495.755,Z 333.733,A -85,B 0,C 180,E1 -6349.954,E2 -6349.954} C_VEL
LIN {X 0,Y 495.727,Z 333.732,A -85,B 0,C 180,E1 -6352.554,E2 -6352.554} C_VEL
LIN {X 0,Y 495.782,Z 333.725,A -85,B 0,C 180,E1 -6355.458,E2 -6355.458} C_VEL
LIN {X 0,Y 495.756,Z 333.73,A -85,B 0,C 180,E1 -6358.365,E2 -6358.365} C_VEL
LIN {X 0,Y 495.764,Z 333.726,A -85,B 0,C 180,E1 -6360.777,E2 -6360.777} C_VEL
LIN {X 0,Y 495.105,Z 333.811,A -85,B 0,C 180,E1 -6361.456,E2 -6361.456} C_VEL
LIN {X 0,Y 492.247,Z 334.165,A -85,B 0,C 180,E1 -6362.558,E2 -6362.558} C_VEL
LIN {X 0,Y 489.838,Z 334.466,A -85,B 0,C 180,E1 -6363.447,E2 -6363.447} C_VEL
LIN {X 0,Y 488.821,Z 334.596,A -85,B 0,C 180,E1 -6364.133,E2 -6364.133} C_VEL
LIN {X 0,Y 488.748,Z 334.601,A -85,B 0,C 180,E1 -6364.366,E2 -6364.366} C_VEL
LIN {X 0,Y 488.729,Z 334.603,A -85,B 0,C 180,E1 -6367.154,E2 -6367.154} C_VEL
LIN {X 0,Y 488.73,Z 334.61,A -85,B 0,C 180,E1 -6369.811,E2 -6369.811} C_VEL
LIN {X 0,Y 488.736,Z 334.602,A -85,B 0,C 180,E1 -6372.424,E2 -6372.424} C_VEL
LIN {X 0,Y 488.764,Z 334.598,A -85,B 0,C 180,E1 -6375,E2 -6375} C_VEL
LIN {X 0,Y 488.808,Z 334.593,A -85,B 0,C 180,E1 -6378.388,E2 -6378.388} C_VEL
LIN {X 0,Y 488.821,Z 334.598,A -85,B 0,C 180,E1 -6381.734,E2 -6381.734} C_VEL
LIN {X 0,Y 488.861,Z 334.587,A -85,B 0,C 180,E1 -6384.224,E2 -6384.224} C_VEL
LIN {X 0,Y 488.965,Z 334.581,A -85,B 0,C 180,E1 -6387.529,E2 -6387.529} C_VEL
LIN {X 0,Y 488.958,Z 334.574,A -85,B 0,C 180,E1 -6390.824,E2 -6390.824} C_VEL
LIN {X 0,Y 488.965,Z 334.572,A -85,B 0,C 180,E1 -6392.471,E2 -6392.471} C_VEL
LIN {X 0,Y 488.851,Z 334.591,A -85,B 0,C 180,E1 -6395.776,E2 -6395.776} C_VEL
LIN {X 0,Y 488.82,Z 334.591,A -85,B 0,C 180,E1 -6398.266,E2 -6398.266} C_VEL
LIN {X 0,Y 488.808,Z 334.597,A -85,B 0,C 180,E1 -6401.612,E2 -6401.612} C_VEL
LIN {X 0,Y 488.764,Z 334.601,A -85,B 0,C 180,E1 -6405,E2 -6405} C_VEL
LIN {X 0,Y 488.756,Z 334.599,A -85,B 0,C 180,E1 -6408.442,E2 -6408.442} C_VEL
LIN {X 0,Y 488.708,Z 334.611,A -85,B 0,C 180,E1 -6411.07,E2 -6411.07} C_VEL
LIN {X 0,Y 488.694,Z 334.608,A -85,B 0,C 180,E1 -6413.745,E2 -6413.745} C_VEL
LIN {X 0,Y 488.799,Z 334.599,A -85,B 0,C 180,E1 -6416.945,E2 -6416.945} C_VEL
LIN {X 0,Y 488.709,Z 334.605,A -85,B 0,C 180,E1 -6420.362,E2 -6420.362} C_VEL
LIN {X 0,Y 488.735,Z 334.604,A -85,B 0,C 180,E1 -6423.484,E2 -6423.484} C_VEL
LIN {X 0,Y 488.688,Z 334.608,A -85,B 0,C 180,E1 -6426.355,E2 -6426.355} C_VEL
LIN {X 0,Y 488.746,Z 334.606,A -85,B 0,C 180,E1 -6429.249,E2 -6429.249} C_VEL
LIN {X 0,Y 488.73,Z 334.607,A -85,B 0,C 180,E1 -6432.52,E2 -6432.52} C_VEL
LIN {X 0,Y 488.707,Z 334.612,A -85,B 0,C 180,E1 -6435.198,E2 -6435.198} C_VEL
LIN {X 0,Y 488.761,Z 334.783,A -85,B 0,C 180,E1 -6438.063,E2 -6438.063} C_VEL
LIN {X 0,Y 489.093,Z 336.12,A -85,B 0,C 180,E1 -6438.224,E2 -6438.224} C_VEL
LIN {X 0,Y 490.833,Z 342.448,A -85,B 0,C 180,E1 -6438.609,E2 -6438.609} C_VEL
LIN {X 0,Y 490.577,Z 354.348,A -85,B 0,C 180,E1 -6439.342,E2 -6439.342} C_VEL
LIN {X 0,Y 490.145,Z 365.492,A -85,B 0,C 180,E1 -6440.216,E2 -6440.216} C_VEL
LIN {X 0,Y 489.784,Z 375.923,A -85,B 0,C 180,E1 -6441.246,E2 -6441.246} C_VEL
LIN {X 0,Y 489.394,Z 385.458,A -85,B 0,C 180,E1 -6442.411,E2 -6442.411} C_VEL
LIN {X 0,Y 489.092,Z 393.13,A -85,B 0,C 180,E1 -6443.578,E2 -6443.578} C_VEL
LIN {X 0,Y 488.856,Z 400.1,A -85,B 0,C 180,E1 -6444.896,E2 -6444.896} C_VEL
LIN {X 0,Y 488.611,Z 405.767,A -85,B 0,C 180,E1 -6446.255,E2 -6446.255} C_VEL
LIN {X 0,Y 488.485,Z 409.295,A -85,B 0,C 180,E1 -6447.349,E2 -6447.349} C_VEL
LIN {X 0,Y 488.426,Z 412.78,A -85,B 0,C 180,E1 -6448.801,E2 -6448.801} C_VEL
LIN {X 0,Y 488.339,Z 414.333,A -85,B 0,C 180,E1 -6449.754,E2 -6449.754} C_VEL
LIN {X 0,Y 488.295,Z 415.392,A -85,B 0,C 180,E1 -6450.701,E2 -6450.701} C_VEL
LIN {X 0,Y 488.297,Z 415.88,A -85,B 0,C 180,E1 -6451.643,E2 -6451.643} C_VEL
LIN {X 0,Y 488.289,Z 415.646,A -85,B 0,C 180,E1 -6453.17,E2 -6453.17} C_VEL
LIN {X 0,Y 488.367,Z 414.437,A -85,B 0,C 180,E1 -6454.423,E2 -6454.423} C_VEL
LIN {X 0,Y 488.453,Z 412.99,A -85,B 0,C 180,E1 -6455.338,E2 -6455.338} C_VEL
LIN {X 0,Y 488.602,Z 409.921,A -85,B 0,C 180,E1 -6456.674,E2 -6456.674} C_VEL
LIN {X 0,Y 488.772,Z 405.527,A -85,B 0,C 180,E1 -6458.047,E2 -6458.047} C_VEL
LIN {X 0,Y 489.006,Z 399.536,A -85,B 0,C 180,E1 -6459.464,E2 -6459.464} C_VEL
LIN {X 0,Y 489.302,Z 392.799,A -85,B 0,C 180,E1 -6460.71,E2 -6460.71} C_VEL
LIN {X 0,Y 489.604,Z 385.465,A -85,B 0,C 180,E1 -6461.808,E2 -6461.808} C_VEL
LIN {X 0,Y 489.954,Z 376.543,A -85,B 0,C 180,E1 -6462.899,E2 -6462.899} C_VEL
LIN {X 0,Y 490.309,Z 367.434,A -85,B 0,C 180,E1 -6463.81,E2 -6463.81} C_VEL
LIN {X 0,Y 490.679,Z 357.32,A -85,B 0,C 180,E1 -6464.634,E2 -6464.634} C_VEL
LIN {X 0,Y 491.006,Z 345.597,A -85,B 0,C 180,E1 -6465.388,E2 -6465.388} C_VEL
LIN {X 0,Y 490.788,Z 342.056,A -85,B 0,C 180,E1 -6465.593,E2 -6465.593} C_VEL
LIN {X 0,Y 488.866,Z 335.305,A -85,B 0,C 180,E1 -6466.013,E2 -6466.013} C_VEL
LIN {X 0,Y 488.759,Z 334.624,A -85,B 0,C 180,E1 -6466.222,E2 -6466.222} C_VEL
LIN {X 0,Y 488.818,Z 334.596,A -85,B 0,C 180,E1 -6468.388,E2 -6468.388} C_VEL
LIN {X 0,Y 488.807,Z 334.598,A -85,B 0,C 180,E1 -6471.733,E2 -6471.733} C_VEL
LIN {X 0,Y 488.836,Z 334.592,A -85,B 0,C 180,E1 -6474.224,E2 -6474.224} C_VEL
LIN {X 0,Y 488.948,Z 334.582,A -85,B 0,C 180,E1 -6477.529,E2 -6477.529} C_VEL
LIN {X 0,Y 488.955,Z 334.577,A -85,B 0,C 180,E1 -6480,E2 -6480} C_VEL
LIN {X 0,Y 488.947,Z 334.577,A -85,B 0,C 180,E1 -6482.471,E2 -6482.471} C_VEL
LIN {X 0,Y 488.834,Z 334.592,A -85,B 0,C 180,E1 -6485.776,E2 -6485.776} C_VEL
LIN {X 0,Y 488.774,Z 334.597,A -85,B 0,C 180,E1 -6488.267,E2 -6488.267} C_VEL
LIN {X 0,Y 488.794,Z 334.597,A -85,B 0,C 180,E1 -6491.613,E2 -6491.613} C_VEL
LIN {X 0,Y 488.751,Z 334.608,A -85,B 0,C 180,E1 -6495.001,E2 -6495.001} C_VEL
LIN {X 0,Y 488.736,Z 334.601,A -85,B 0,C 180,E1 -6498.443,E2 -6498.443} C_VEL
LIN {X 0,Y 488.697,Z 334.611,A -85,B 0,C 180,E1 -6501.071,E2 -6501.071} C_VEL
LIN {X 0,Y 488.672,Z 334.609,A -85,B 0,C 180,E1 -6503.747,E2 -6503.747} C_VEL
LIN {X 0,Y 488.782,Z 334.602,A -85,B 0,C 180,E1 -6506.944,E2 -6506.944} C_VEL
LIN {X 0,Y 488.699,Z 334.609,A -85,B 0,C 180,E1 -6510.363,E2 -6510.363} C_VEL
LIN {X 0,Y 488.721,Z 334.606,A -85,B 0,C 180,E1 -6513.484,E2 -6513.484} C_VEL
LIN {X 0,Y 488.674,Z 334.613,A -85,B 0,C 180,E1 -6516.355,E2 -6516.355} C_VEL
LIN {X 0,Y 488.686,Z 334.612,A -85,B 0,C 180,E1 -6519.256,E2 -6519.256} C_VEL
LIN {X 0,Y 488.66,Z 334.619,A -85,B 0,C 180,E1 -6522.529,E2 -6522.529} C_VEL
LIN {X 0,Y 488.696,Z 334.612,A -85,B 0,C 180,E1 -6525.198,E2 -6525.198} C_VEL
LIN {X 0,Y 488.667,Z 334.618,A -85,B 0,C 180,E1 -6528.581,E2 -6528.581} C_VEL
LIN {X 0,Y 488.717,Z 334.798,A -85,B 0,C 180,E1 -6531.017,E2 -6531.017} C_VEL
LIN {X 0,Y 490.349,Z 343.201,A -85,B 0,C 180,E1 -6533.382,E2 -6533.382} C_VEL
LIN {X 0,Y 490.539,Z 347.298,A -85,B 0,C 180,E1 -6534.447,E2 -6534.447} C_VEL
LIN {X 0,Y 489.811,Z 362.758,A -85,B 0,C 180,E1 -6538.177,E2 -6538.177} C_VEL
LIN {X 0,Y 489.51,Z 375.615,A -85,B 0,C 180,E1 -6541.139,E2 -6541.139} C_VEL
LIN {X 0,Y 489.231,Z 389.621,A -85,B 0,C 180,E1 -6544.244,E2 -6544.244} C_VEL
LIN {X 0,Y 488.956,Z 404.233,A -85,B 0,C 180,E1 -6547.389,E2 -6547.389} C_VEL
LIN {X 0,Y 488.755,Z 418.82,A -85,B 0,C 180,E1 -6550.469,E2 -6550.469} C_VEL
LIN {X 0,Y 488.585,Z 432.349,A -85,B 0,C 180,E1 -6553.281,E2 -6553.281} C_VEL
LIN {X 0,Y 488.458,Z 441.814,A -85,B 0,C 180,E1 -6555.204,E2 -6555.204} C_VEL
LIN {X 0,Y 488.541,Z 443.544,A -85,B 0,C 180,E1 -6555.286,E2 -6555.286} C_VEL
LIN {X 0,Y 489.784,Z 457.701,A -85,B 0,C 180,E1 -6555.669,E2 -6555.669} C_VEL
LIN {X 0,Y 490.448,Z 463.993,A -85,B 0,C 180,E1 -6555.901,E2 -6555.901} C_VEL
LIN {X 0,Y 490.083,Z 476.013,A -85,B 0,C 180,E1 -6556.419,E2 -6556.419} C_VEL
LIN {X 0,Y 489.732,Z 487.49,A -85,B 0,C 180,E1 -6557.074,E2 -6557.074} C_VEL
LIN {X 0,Y 489.4,Z 498.34,A -85,B 0,C 180,E1 -6557.854,E2 -6557.854} C_VEL
LIN {X 0,Y 488.993,Z 509.147,A -85,B 0,C 180,E1 -6558.812,E2 -6558.812} C_VEL
LIN {X 0,Y 488.645,Z 518.685,A -85,B 0,C 180,E1 -6559.853,E2 -6559.853} C_VEL
LIN {X 0,Y 488.419,Z 527.939,A -85,B 0,C 180,E1 -6561.102,E2 -6561.102} C_VEL
LIN {X 0,Y 488.294,Z 535.433,A -85,B 0,C 180,E1 -6562.349,E2 -6562.349} C_VEL
LIN {X 0,Y 488.193,Z 541.674,A -85,B 0,C 180,E1 -6563.649,E2 -6563.649} C_VEL
LIN {X 0,Y 488.163,Z 546.829,A -85,B 0,C 180,E1 -6565.045,E2 -6565.045} C_VEL
LIN {X 0,Y 488.186,Z 549.235,A -85,B 0,C 180,E1 -6565.872,E2 -6565.872} C_VEL
LIN {X 0,Y 488.122,Z 551.189,A -85,B 0,C 180,E1 -6566.698,E2 -6566.698} C_VEL
LIN {X 0,Y 488.104,Z 552.662,A -85,B 0,C 180,E1 -6567.524,E2 -6567.524} C_VEL
LIN {X 0,Y 488.124,Z 554.374,A -85,B 0,C 180,E1 -6569.175,E2 -6569.175} C_VEL
LIN {X 0,Y 488.111,Z 554.621,A -85,B 0,C 180,E1 -6570,E2 -6570} C_VEL
LIN {X 0,Y 488.123,Z 554.418,A -85,B 0,C 180,E1 -6570.825,E2 -6570.825} C_VEL
LIN {X 0,Y 488.088,Z 552.803,A -85,B 0,C 180,E1 -6572.476,E2 -6572.476} C_VEL
LIN {X 0,Y 488.103,Z 551.374,A -85,B 0,C 180,E1 -6573.302,E2 -6573.302} C_VEL
LIN {X 0,Y 488.1,Z 548.374,A -85,B 0,C 180,E1 -6574.542,E2 -6574.542} C_VEL
LIN {X 0,Y 488.202,Z 543.256,A -85,B 0,C 180,E1 -6576.051,E2 -6576.051} C_VEL
LIN {X 0,Y 488.22,Z 537.004,A -85,B 0,C 180,E1 -6577.444,E2 -6577.444} C_VEL
LIN {X 0,Y 488.361,Z 529.924,A -85,B 0,C 180,E1 -6578.691,E2 -6578.691} C_VEL
LIN {X 0,Y 488.593,Z 521.078,A -85,B 0,C 180,E1 -6579.939,E2 -6579.939} C_VEL
LIN {X 0,Y 488.988,Z 511.09,A -85,B 0,C 180,E1 -6581.083,E2 -6581.083} C_VEL
LIN {X 0,Y 489.408,Z 500.941,A -85,B 0,C 180,E1 -6582.018,E2 -6582.018} C_VEL
LIN {X 0,Y 489.682,Z 490.374,A -85,B 0,C 180,E1 -6582.811,E2 -6582.811} C_VEL
LIN {X 0,Y 490.089,Z 479.278,A -85,B 0,C 180,E1 -6583.475,E2 -6583.475} C_VEL
LIN {X 0,Y 490.469,Z 466.859,A -85,B 0,C 180,E1 -6584.046,E2 -6584.046} C_VEL
LIN {X 0,Y 490.334,Z 461.025,A -85,B 0,C 180,E1 -6584.261,E2 -6584.261} C_VEL
LIN {X 0,Y 489.083,Z 449.924,A -85,B 0,C 180,E1 -6584.604,E2 -6584.604} C_VEL
LIN {X 0,Y 488.479,Z 443.73,A -85,B 0,C 180,E1 -6584.769,E2 -6584.769} C_VEL
LIN {X 0,Y 488.555,Z 440.071,A -85,B 0,C 180,E1 -6585.46,E2 -6585.46} C_VEL
LIN {X 0,Y 488.783,Z 425.158,A -85,B 0,C 180,E1 -6588.658,E2 -6588.658} C_VEL
LIN {X 0,Y 489.091,Z 410.033,A -85,B 0,C 180,E1 -6591.938,E2 -6591.938} C_VEL
LIN {X 0,Y 489.447,Z 396.547,A -85,B 0,C 180,E1 -6594.924,E2 -6594.924} C_VEL
LIN {X 0,Y 489.824,Z 383.831,A -85,B 0,C 180,E1 -6597.794,E2 -6597.794} C_VEL
LIN {X 0,Y 490.255,Z 371.41,A -85,B 0,C 180,E1 -6600.669,E2 -6600.669} C_VEL
LIN {X 0,Y 490.939,Z 355.637,A -85,B 0,C 180,E1 -6604.433,E2 -6604.433} C_VEL
LIN {X 0,Y 491.296,Z 348.021,A -85,B 0,C 180,E1 -6606.306,E2 -6606.306} C_VEL
LIN {X 0,Y 489.686,Z 339.463,A -85,B 0,C 180,E1 -6608.6,E2 -6608.6} C_VEL
LIN {X 0,Y 488.704,Z 334.686,A -85,B 0,C 180,E1 -6609.988,E2 -6609.988} C_VEL
LIN {X 0,Y 488.66,Z 334.617,A -85,B 0,C 180,E1 -6612.82,E2 -6612.82} C_VEL
LIN {X 0,Y 488.683,Z 334.612,A -85,B 0,C 180,E1 -6615.977,E2 -6615.977} C_VEL
LIN {X 0,Y 488.66,Z 334.611,A -85,B 0,C 180,E1 -6618.579,E2 -6618.579} C_VEL
LIN {X 0,Y 488.691,Z 334.61,A -85,B 0,C 180,E1 -6620.948,E2 -6620.948} C_VEL
LIN {X 0,Y 488.669,Z 334.611,A -85,B 0,C 180,E1 -6623.867,E2 -6623.867} C_VEL
LIN {X 0,Y 488.727,Z 334.605,A -85,B 0,C 180,E1 -6626.876,E2 -6626.876} C_VEL
LIN {X 0,Y 488.714,Z 334.606,A -85,B 0,C 180,E1 -6629.78,E2 -6629.78} C_VEL
LIN {X 0,Y 488.783,Z 334.602,A -85,B 0,C 180,E1 -6633.056,E2 -6633.056} C_VEL
LIN {X 0,Y 488.665,Z 334.61,A -85,B 0,C 180,E1 -6636.253,E2 -6636.253} C_VEL
LIN {X 0,Y 488.737,Z 334.609,A -85,B 0,C 180,E1 -6639.175,E2 -6639.175} C_VEL
LIN {X 0,Y 488.739,Z 334.602,A -85,B 0,C 180,E1 -6641.631,E2 -6641.631} C_VEL
LIN {X 0,Y 488.751,Z 334.608,A -85,B 0,C 180,E1 -6644.999,E2 -6644.999} C_VEL
LIN {X 0,Y 488.794,Z 334.595,A -85,B 0,C 180,E1 -6648.387,E2 -6648.387} C_VEL
LIN {X 0,Y 488.774,Z 334.597,A -85,B 0,C 180,E1 -6651.733,E2 -6651.733} C_VEL
LIN {X 0,Y 488.834,Z 334.59,A -85,B 0,C 180,E1 -6654.224,E2 -6654.224} C_VEL
LIN {X 0,Y 488.947,Z 334.576,A -85,B 0,C 180,E1 -6657.529,E2 -6657.529} C_VEL
LIN {X 0,Y 488.955,Z 334.574,A -85,B 0,C 180,E1 -6660,E2 -6660} C_VEL
LIN {X 0,Y 488.948,Z 334.579,A -85,B 0,C 180,E1 -6662.471,E2 -6662.471} C_VEL
LIN {X 0,Y 488.835,Z 334.589,A -85,B 0,C 180,E1 -6665.776,E2 -6665.776} C_VEL
LIN {X 0,Y 488.807,Z 334.595,A -85,B 0,C 180,E1 -6668.267,E2 -6668.267} C_VEL
LIN {X 0,Y 488.796,Z 334.594,A -85,B 0,C 180,E1 -6671.613,E2 -6671.613} C_VEL
LIN {X 0,Y 488.754,Z 334.602,A -85,B 0,C 180,E1 -6675.001,E2 -6675.001} C_VEL
LIN {X 0,Y 488.745,Z 334.607,A -85,B 0,C 180,E1 -6678.443,E2 -6678.443} C_VEL
LIN {X 0,Y 488.703,Z 334.607,A -85,B 0,C 180,E1 -6681.071,E2 -6681.071} C_VEL
LIN {X 0,Y 488.692,Z 334.607,A -85,B 0,C 180,E1 -6683.746,E2 -6683.746} C_VEL
LIN {X 0,Y 488.783,Z 334.597,A -85,B 0,C 180,E1 -6686.944,E2 -6686.944} C_VEL
LIN {X 0,Y 488.726,Z 334.609,A -85,B 0,C 180,E1 -6690.219,E2 -6690.219} C_VEL
LIN {X 0,Y 488.728,Z 334.602,A -85,B 0,C 180,E1 -6693.485,E2 -6693.485} C_VEL
LIN {X 0,Y 488.68,Z 334.616,A -85,B 0,C 180,E1 -6696.356,E2 -6696.356} C_VEL
LIN {X 0,Y 488.731,Z 334.602,A -85,B 0,C 180,E1 -6699.251,E2 -6699.251} C_VEL
LIN {X 0,Y 488.706,Z 334.606,A -85,B 0,C 180,E1 -6701.601,E2 -6701.601} C_VEL
LIN {X 0,Y 488.707,Z 334.606,A -85,B 0,C 180,E1 -6704.802,E2 -6704.802} C_VEL
LIN {X 0,Y 488.69,Z 334.608,A -85,B 0,C 180,E1 -6707.476,E2 -6707.476} C_VEL
LIN {X 0,Y 488.729,Z 334.605,A -85,B 0,C 180,E1 -6709.677,E2 -6709.677} C_VEL
LIN {X 0,Y 488.679,Z 334.608,A -85,B 0,C 180,E1 -6712.842,E2 -6712.842} C_VEL
LIN {X 0,Y 488.732,Z 334.608,A -85,B 0,C 180,E1 -6715.888,E2 -6715.888} C_VEL
LIN {X 0,Y 488.694,Z 334.606,A -85,B 0,C 180,E1 -6718.821,E2 -6718.821} C_VEL
LIN {X 0,Y 488.747,Z 334.604,A -85,B 0,C 180,E1 -6721.672,E2 -6721.672} C_VEL
LIN {X 0,Y 488.748,Z 334.601,A -85,B 0,C 180,E1 -6724.366,E2 -6724.366} C_VEL
LIN {X 0,Y 488.102,Z 334.685,A -85,B 0,C 180,E1 -6725.053,E2 -6725.053} C_VEL
LIN {X 0,Y 485.233,Z 335.047,A -85,B 0,C 180,E1 -6726.17,E2 -6726.17} C_VEL
LIN {X 0,Y 482.786,Z 335.351,A -85,B 0,C 180,E1 -6727.07,E2 -6727.07} C_VEL
LIN {X 0,Y 481.728,Z 335.481,A -85,B 0,C 180,E1 -6727.765,E2 -6727.765} C_VEL
LIN {X 0,Y 481.639,Z 335.488,A -85,B 0,C 180,E1 -6728.001,E2 -6728.001} C_VEL
LIN {X 0,Y 481.709,Z 335.478,A -85,B 0,C 180,E1 -6730.394,E2 -6730.394} C_VEL
LIN {X 0,Y 481.693,Z 335.479,A -85,B 0,C 180,E1 -6733.034,E2 -6733.034} C_VEL
LIN {X 0,Y 481.693,Z 335.486,A -85,B 0,C 180,E1 -6735.639,E2 -6735.639} C_VEL
LIN {X 0,Y 481.753,Z 335.473,A -85,B 0,C 180,E1 -6738.215,E2 -6738.215} C_VEL
LIN {X 0,Y 481.766,Z 335.477,A -85,B 0,C 180,E1 -6741.612,E2 -6741.612} C_VEL
LIN {X 0,Y 481.822,Z 335.464,A -85,B 0,C 180,E1 -6744.14,E2 -6744.14} C_VEL
LIN {X 0,Y 481.932,Z 335.456,A -85,B 0,C 180,E1 -6747.493,E2 -6747.493} C_VEL
LIN {X 0,Y 481.909,Z 335.452,A -85,B 0,C 180,E1 -6750.836,E2 -6750.836} C_VEL
LIN {X 0,Y 481.932,Z 335.449,A -85,B 0,C 180,E1 -6752.507,E2 -6752.507} C_VEL
LIN {X 0,Y 481.812,Z 335.467,A -85,B 0,C 180,E1 -6755.86,E2 -6755.86} C_VEL
LIN {X 0,Y 481.765,Z 335.469,A -85,B 0,C 180,E1 -6758.388,E2 -6758.388} C_VEL
LIN {X 0,Y 481.753,Z 335.474,A -85,B 0,C 180,E1 -6761.785,E2 -6761.785} C_VEL
LIN {X 0,Y 481.745,Z 335.479,A -85,B 0,C 180,E1 -6765.224,E2 -6765.224} C_VEL
LIN {X 0,Y 481.714,Z 335.477,A -85,B 0,C 180,E1 -6768.721,E2 -6768.721} C_VEL
LIN {X 0,Y 481.648,Z 335.49,A -85,B 0,C 180,E1 -6771.394,E2 -6771.394} C_VEL
LIN {X 0,Y 481.678,Z 335.48,A -85,B 0,C 180,E1 -6774.112,E2 -6774.112} C_VEL
LIN {X 0,Y 481.752,Z 335.479,A -85,B 0,C 180,E1 -6777.14,E2 -6777.14} C_VEL
LIN {X 0,Y 481.678,Z 335.481,A -85,B 0,C 180,E1 -6779.74,E2 -6779.74} C_VEL
LIN {X 0,Y 481.672,Z 335.484,A -85,B 0,C 180,E1 -6782.673,E2 -6782.673} C_VEL
LIN {X 0,Y 481.642,Z 335.486,A -85,B 0,C 180,E1 -6785.708,E2 -6785.708} C_VEL
LIN {X 0,Y 481.717,Z 335.481,A -85,B 0,C 180,E1 -6789.354,E2 -6789.354} C_VEL
LIN {X 0,Y 481.672,Z 335.484,A -85,B 0,C 180,E1 -6792.157,E2 -6792.157} C_VEL
LIN {X 0,Y 481.656,Z 335.489,A -85,B 0,C 180,E1 -6794.456,E2 -6794.456} C_VEL
LIN {X 0,Y 481.727,Z 335.604,A -85,B 0,C 180,E1 -6797.848,E2 -6797.848} C_VEL
LIN {X 0,Y 481.954,Z 336.678,A -85,B 0,C 180,E1 -6798.004,E2 -6798.004} C_VEL
LIN {X 0,Y 483.846,Z 343.369,A -85,B 0,C 180,E1 -6798.42,E2 -6798.42} C_VEL
LIN {X 0,Y 483.709,Z 355.271,A -85,B 0,C 180,E1 -6799.169,E2 -6799.169} C_VEL
LIN {X 0,Y 483.305,Z 365.228,A -85,B 0,C 180,E1 -6799.949,E2 -6799.949} C_VEL
LIN {X 0,Y 482.899,Z 375.871,A -85,B 0,C 180,E1 -6800.99,E2 -6800.99} C_VEL
LIN {X 0,Y 482.531,Z 384.765,A -85,B 0,C 180,E1 -6802.063,E2 -6802.063} C_VEL
LIN {X 0,Y 482.186,Z 393.134,A -85,B 0,C 180,E1 -6803.303,E2 -6803.303} C_VEL
LIN {X 0,Y 481.885,Z 400.847,A -85,B 0,C 180,E1 -6804.756,E2 -6804.756} C_VEL
LIN {X 0,Y 481.673,Z 405.393,A -85,B 0,C 180,E1 -6805.824,E2 -6805.824} C_VEL
LIN {X 0,Y 481.483,Z 410.338,A -85,B 0,C 180,E1 -6807.311,E2 -6807.311} C_VEL
LIN {X 0,Y 481.429,Z 412.793,A -85,B 0,C 180,E1 -6808.296,E2 -6808.296} C_VEL
LIN {X 0,Y 481.361,Z 414.974,A -85,B 0,C 180,E1 -6809.473,E2 -6809.473} C_VEL
LIN {X 0,Y 481.281,Z 415.944,A -85,B 0,C 180,E1 -6810.232,E2 -6810.232} C_VEL
LIN {X 0,Y 481.277,Z 416.707,A -85,B 0,C 180,E1 -6811.191,E2 -6811.191} C_VEL
LIN {X 0,Y 481.277,Z 416.965,A -85,B 0,C 180,E1 -6812.141,E2 -6812.141} C_VEL
LIN {X 0,Y 481.269,Z 416.711,A -85,B 0,C 180,E1 -6813.083,E2 -6813.083} C_VEL
LIN {X 0,Y 481.332,Z 415.992,A -85,B 0,C 180,E1 -6814.021,E2 -6814.021} C_VEL
LIN {X 0,Y 481.391,Z 414.746,A -85,B 0,C 180,E1 -6814.952,E2 -6814.952} C_VEL
LIN {X 0,Y 481.565,Z 411.97,A -85,B 0,C 180,E1 -6816.338,E2 -6816.338} C_VEL
LIN {X 0,Y 481.725,Z 408.053,A -85,B 0,C 180,E1 -6817.708,E2 -6817.708} C_VEL
LIN {X 0,Y 482.012,Z 402.1,A -85,B 0,C 180,E1 -6819.238,E2 -6819.238} C_VEL
LIN {X 0,Y 482.294,Z 394.981,A -85,B 0,C 180,E1 -6820.64,E2 -6820.64} C_VEL
LIN {X 0,Y 482.626,Z 387.904,A -85,B 0,C 180,E1 -6821.755,E2 -6821.755} C_VEL
LIN {X 0,Y 483.001,Z 379.289,A -85,B 0,C 180,E1 -6822.863,E2 -6822.863} C_VEL
LIN {X 0,Y 483.429,Z 368.626,A -85,B 0,C 180,E1 -6823.965,E2 -6823.965} C_VEL
LIN {X 0,Y 483.843,Z 357.985,A -85,B 0,C 180,E1 -6824.843,E2 -6824.843} C_VEL
LIN {X 0,Y 484.196,Z 346.139,A -85,B 0,C 180,E1 -6825.607,E2 -6825.607} C_VEL
LIN {X 0,Y 483.773,Z 342.832,A -85,B 0,C 180,E1 -6825.809,E2 -6825.809} C_VEL
LIN {X 0,Y 481.822,Z 336.178,A -85,B 0,C 180,E1 -6826.235,E2 -6826.235} C_VEL
LIN {X 0,Y 481.719,Z 335.501,A -85,B 0,C 180,E1 -6826.447,E2 -6826.447} C_VEL
LIN {X 0,Y 481.707,Z 335.484,A -85,B 0,C 180,E1 -6829.067,E2 -6829.067} C_VEL
LIN {X 0,Y 481.818,Z 335.466,A -85,B 0,C 180,E1 -6832.457,E2 -6832.457} C_VEL
LIN {X 0,Y 481.767,Z 335.475,A -85,B 0,C 180,E1 -6834.979,E2 -6834.979} C_VEL
LIN {X 0,Y 481.915,Z 335.459,A -85,B 0,C 180,E1 -6837.493,E2 -6837.493} C_VEL
LIN {X 0,Y 481.895,Z 335.458,A -85,B 0,C 180,E1 -6840.836,E2 -6840.836} C_VEL
LIN {X 0,Y 481.914,Z 335.453,A -85,B 0,C 180,E1 -6842.508,E2 -6842.508} C_VEL
LIN {X 0,Y 481.795,Z 335.468,A -85,B 0,C 180,E1 -6845.861,E2 -6845.861} C_VEL
LIN {X 0,Y 481.729,Z 335.475,A -85,B 0,C 180,E1 -6848.389,E2 -6848.389} C_VEL
LIN {X 0,Y 481.74,Z 335.474,A -85,B 0,C 180,E1 -6851.785,E2 -6851.785} C_VEL
LIN {X 0,Y 481.732,Z 335.481,A -85,B 0,C 180,E1 -6855.225,E2 -6855.225} C_VEL
LIN {X 0,Y 481.698,Z 335.481,A -85,B 0,C 180,E1 -6858.722,E2 -6858.722} C_VEL
LIN {X 0,Y 481.635,Z 335.491,A -85,B 0,C 180,E1 -6861.395,E2 -6861.395} C_VEL
LIN {X 0,Y 481.657,Z 335.483,A -85,B 0,C 180,E1 -6864.114,E2 -6864.114} C_VEL
LIN {X 0,Y 481.737,Z 335.48,A -85,B 0,C 180,E1 -6867.139,E2 -6867.139} C_VEL
LIN {X 0,Y 481.669,Z 335.484,A -85,B 0,C 180,E1 -6869.742,E2 -6869.742} C_VEL
LIN {X 0,Y 481.662,Z 335.49,A -85,B 0,C 180,E1 -6872.675,E2 -6872.675} C_VEL
LIN {X 0,Y 481.628,Z 335.489,A -85,B 0,C 180,E1 -6875.71,E2 -6875.71} C_VEL
LIN {X 0,Y 481.659,Z 335.49,A -85,B 0,C 180,E1 -6878.86,E2 -6878.86} C_VEL
LIN {X 0,Y 481.618,Z 335.492,A -85,B 0,C 180,E1 -6882.164,E2 -6882.164} C_VEL
LIN {X 0,Y 481.648,Z 335.488,A -85,B 0,C 180,E1 -6885.543,E2 -6885.543} C_VEL
LIN {X 0,Y 481.624,Z 335.493,A -85,B 0,C 180,E1 -6888.956,E2 -6888.956} C_VEL
LIN {X 0,Y 481.666,Z 335.647,A -85,B 0,C 180,E1 -6890.727,E2 -6890.727} C_VEL
LIN {X 0,Y 483.483,Z 344.996,A -85,B 0,C 180,E1 -6893.418,E2 -6893.418} C_VEL
LIN {X 0,Y 483.59,Z 349.035,A -85,B 0,C 180,E1 -6894.474,E2 -6894.474} C_VEL
LIN {X 0,Y 482.833,Z 363.281,A -85,B 0,C 180,E1 -6897.987,E2 -6897.987} C_VEL
LIN {X 0,Y 482.527,Z 374.647,A -85,B 0,C 180,E1 -6900.664,E2 -6900.664} C_VEL
LIN {X 0,Y 482.217,Z 388.648,A -85,B 0,C 180,E1 -6903.841,E2 -6903.841} C_VEL
LIN {X 0,Y 481.907,Z 403.176,A -85,B 0,C 180,E1 -6907.039,E2 -6907.039} C_VEL
LIN {X 0,Y 481.69,Z 417.748,A -85,B 0,C 180,E1 -6910.171,E2 -6910.171} C_VEL
LIN {X 0,Y 481.493,Z 431.226,A -85,B 0,C 180,E1 -6913.027,E2 -6913.027} C_VEL
LIN {X 0,Y 481.405,Z 440.692,A -85,B 0,C 180,E1 -6914.982,E2 -6914.982} C_VEL
LIN {X 0,Y 481.524,Z 442.58,A -85,B 0,C 180,E1 -6915.067,E2 -6915.067} C_VEL
LIN {X 0,Y 482.716,Z 457.325,A -85,B 0,C 180,E1 -6915.482,E2 -6915.482} C_VEL
LIN {X 0,Y 483.471,Z 464.212,A -85,B 0,C 180,E1 -6915.747,E2 -6915.747} C_VEL
LIN {X 0,Y 483.057,Z 476.779,A -85,B 0,C 180,E1 -6916.325,E2 -6916.325} C_VEL
LIN {X 0,Y 482.645,Z 488.966,A -85,B 0,C 180,E1 -6917.063,E2 -6917.063} C_VEL
LIN {X 0,Y 482.331,Z 499.646,A -85,B 0,C 180,E1 -6917.878,E2 -6917.878} C_VEL
LIN {X 0,Y 481.917,Z 510.045,A -85,B 0,C 180,E1 -6918.859,E2 -6918.859} C_VEL
LIN {X 0,Y 481.529,Z 519.206,A -85,B 0,C 180,E1 -6919.913,E2 -6919.913} C_VEL
LIN {X 0,Y 481.313,Z 528.216,A -85,B 0,C 180,E1 -6921.181,E2 -6921.181} C_VEL
LIN {X 0,Y 481.201,Z 535.436,A -85,B 0,C 180,E1 -6922.447,E2 -6922.447} C_VEL
LIN {X 0,Y 481.128,Z 540.951,A -85,B 0,C 180,E1 -6923.642,E2 -6923.642} C_VEL
LIN {X 0,Y 481.113,Z 545.781,A -85,B 0,C 180,E1 -6924.972,E2 -6924.972} C_VEL
LIN {X 0,Y 481.127,Z 548.2,A -85,B 0,C 180,E1 -6925.812,E2 -6925.812} C_VEL
LIN {X 0,Y 481.079,Z 550.165,A -85,B 0,C 180,E1 -6926.65,E2 -6926.65} C_VEL
LIN {X 0,Y 481.064,Z 551.646,A -85,B 0,C 180,E1 -6927.488,E2 -6927.488} C_VEL
LIN {X 0,Y 481.109,Z 553.378,A -85,B 0,C 180,E1 -6929.163,E2 -6929.163} C_VEL
LIN {X 0,Y 481.097,Z 553.63,A -85,B 0,C 180,E1 -6930,E2 -6930} C_VEL
LIN {X 0,Y 481.109,Z 553.431,A -85,B 0,C 180,E1 -6930.837,E2 -6930.837} C_VEL
LIN {X 0,Y 481.044,Z 551.821,A -85,B 0,C 180,E1 -6932.512,E2 -6932.512} C_VEL
LIN {X 0,Y 481.057,Z 550.392,A -85,B 0,C 180,E1 -6933.35,E2 -6933.35} C_VEL
LIN {X 0,Y 481.048,Z 547.393,A -85,B 0,C 180,E1 -6934.609,E2 -6934.609} C_VEL
LIN {X 0,Y 481.123,Z 543.326,A -85,B 0,C 180,E1 -6935.869,E2 -6935.869} C_VEL
LIN {X 0,Y 481.12,Z 537.036,A -85,B 0,C 180,E1 -6937.343,E2 -6937.343} C_VEL
LIN {X 0,Y 481.284,Z 530.207,A -85,B 0,C 180,E1 -6938.608,E2 -6938.608} C_VEL
LIN {X 0,Y 481.481,Z 521.718,A -85,B 0,C 180,E1 -6939.875,E2 -6939.875} C_VEL
LIN {X 0,Y 481.866,Z 513.021,A -85,B 0,C 180,E1 -6940.929,E2 -6940.929} C_VEL
LIN {X 0,Y 482.235,Z 503.651,A -85,B 0,C 180,E1 -6941.868,E2 -6941.868} C_VEL
LIN {X 0,Y 482.576,Z 493.238,A -85,B 0,C 180,E1 -6942.725,E2 -6942.725} C_VEL
LIN {X 0,Y 482.988,Z 482.071,A -85,B 0,C 180,E1 -6943.463,E2 -6943.463} C_VEL
LIN {X 0,Y 483.446,Z 469.584,A -85,B 0,C 180,E1 -6944.093,E2 -6944.093} C_VEL
LIN {X 0,Y 483.391,Z 461.854,A -85,B 0,C 180,E1 -6944.403,E2 -6944.403} C_VEL
LIN {X 0,Y 482.183,Z 450.51,A -85,B 0,C 180,E1 -6944.777,E2 -6944.777} C_VEL
LIN {X 0,Y 481.429,Z 442.795,A -85,B 0,C 180,E1 -6944.99,E2 -6944.99} C_VEL
LIN {X 0,Y 481.48,Z 438.89,A -85,B 0,C 180,E1 -6945.767,E2 -6945.767} C_VEL
LIN {X 0,Y 481.75,Z 423.3,A -85,B 0,C 180,E1 -6949.162,E2 -6949.162} C_VEL
LIN {X 0,Y 482.135,Z 408.267,A -85,B 0,C 180,E1 -6952.497,E2 -6952.497} C_VEL
LIN {X 0,Y 482.559,Z 393.175,A -85,B 0,C 180,E1 -6955.907,E2 -6955.907} C_VEL
LIN {X 0,Y 483.001,Z 379.047,A -85,B 0,C 180,E1 -6959.186,E2 -6959.186} C_VEL
LIN {X 0,Y 483.485,Z 366.015,A -85,B 0,C 180,E1 -6962.289,E2 -6962.289} C_VEL
LIN {X 0,Y 484.304,Z 352.332,A -85,B 0,C 180,E1 -6965.644,E2 -6965.644} C_VEL
LIN {X 0,Y 484.297,Z 348.915,A -85,B 0,C 180,E1 -6966.51,E2 -6966.51} C_VEL
LIN {X 0,Y 482.216,Z 338.335,A -85,B 0,C 180,E1 -6969.426,E2 -6969.426} C_VEL
LIN {X 0,Y 481.684,Z 335.563,A -85,B 0,C 180,E1 -6970.263,E2 -6970.263} C_VEL
LIN {X 0,Y 481.617,Z 335.496,A -85,B 0,C 180,E1 -6973.301,E2 -6973.301} C_VEL
LIN {X 0,Y 481.647,Z 335.492,A -85,B 0,C 180,E1 -6975.641,E2 -6975.641} C_VEL
LIN {X 0,Y 481.619,Z 335.491,A -85,B 0,C 180,E1 -6978.954,E2 -6978.954} C_VEL
LIN {X 0,Y 481.645,Z 335.485,A -85,B 0,C 180,E1 -6981.992,E2 -6981.992} C_VEL
LIN {X 0,Y 481.676,Z 335.489,A -85,B 0,C 180,E1 -6985.317,E2 -6985.317} C_VEL
LIN {X 0,Y 481.635,Z 335.486,A -85,B 0,C 180,E1 -6988.311,E2 -6988.311} C_VEL
LIN {X 0,Y 481.69,Z 335.487,A -85,B 0,C 180,E1 -6991.218,E2 -6991.218} C_VEL
LIN {X 0,Y 481.679,Z 335.48,A -85,B 0,C 180,E1 -6994.041,E2 -6994.041} C_VEL
LIN {X 0,Y 481.665,Z 335.486,A -85,B 0,C 180,E1 -6996.811,E2 -6996.811} C_VEL
LIN {X 0,Y 481.685,Z 335.482,A -85,B 0,C 180,E1 -6999.502,E2 -6999.502} C_VEL
LIN {X 0,Y 481.681,Z 335.48,A -85,B 0,C 180,E1 -7002.157,E2 -7002.157} C_VEL
LIN {X 0,Y 481.732,Z 335.479,A -85,B 0,C 180,E1 -7004.775,E2 -7004.775} C_VEL
LIN {X 0,Y 481.74,Z 335.473,A -85,B 0,C 180,E1 -7008.215,E2 -7008.215} C_VEL
LIN {X 0,Y 481.729,Z 335.475,A -85,B 0,C 180,E1 -7011.611,E2 -7011.611} C_VEL
LIN {X 0,Y 481.795,Z 335.466,A -85,B 0,C 180,E1 -7014.139,E2 -7014.139} C_VEL
LIN {X 0,Y 481.914,Z 335.452,A -85,B 0,C 180,E1 -7017.492,E2 -7017.492} C_VEL
LIN {X 0,Y 481.895,Z 335.461,A -85,B 0,C 180,E1 -7020.836,E2 -7020.836} C_VEL
LIN {X 0,Y 481.915,Z 335.456,A -85,B 0,C 180,E1 -7022.507,E2 -7022.507} C_VEL
LIN {X 0,Y 481.796,Z 335.466,A -85,B 0,C 180,E1 -7025.861,E2 -7025.861} C_VEL
LIN {X 0,Y 481.752,Z 335.475,A -85,B 0,C 180,E1 -7028.388,E2 -7028.388} C_VEL
LIN {X 0,Y 481.741,Z 335.473,A -85,B 0,C 180,E1 -7031.785,E2 -7031.785} C_VEL
LIN {X 0,Y 481.734,Z 335.474,A -85,B 0,C 180,E1 -7035.224,E2 -7035.224} C_VEL
LIN {X 0,Y 481.703,Z 335.483,A -85,B 0,C 180,E1 -7038.722,E2 -7038.722} C_VEL
LIN {X 0,Y 481.645,Z 335.484,A -85,B 0,C 180,E1 -7041.395,E2 -7041.395} C_VEL
LIN {X 0,Y 481.673,Z 335.484,A -85,B 0,C 180,E1 -7044.113,E2 -7044.113} C_VEL
LIN {X 0,Y 481.738,Z 335.473,A -85,B 0,C 180,E1 -7047.14,E2 -7047.14} C_VEL
LIN {X 0,Y 481.68,Z 335.481,A -85,B 0,C 180,E1 -7049.741,E2 -7049.741} C_VEL
LIN {X 0,Y 481.665,Z 335.486,A -85,B 0,C 180,E1 -7052.675,E2 -7052.675} C_VEL
LIN {X 0,Y 481.634,Z 335.487,A -85,B 0,C 180,E1 -7055.71,E2 -7055.71} C_VEL
LIN {X 0,Y 481.704,Z 335.477,A -85,B 0,C 180,E1 -7059.354,E2 -7059.354} C_VEL
LIN {X 0,Y 481.643,Z 335.493,A -85,B 0,C 180,E1 -7062.161,E2 -7062.161} C_VEL
LIN {X 0,Y 481.655,Z 335.484,A -85,B 0,C 180,E1 -7065.544,E2 -7065.544} C_VEL
LIN {X 0,Y 481.658,Z 335.491,A -85,B 0,C 180,E1 -7068.087,E2 -7068.087} C_VEL
LIN {X 0,Y 481.667,Z 335.482,A -85,B 0,C 180,E1 -7071.142,E2 -7071.142} C_VEL
LIN {X 0,Y 481.665,Z 335.482,A -85,B 0,C 180,E1 -7074.796,E2 -7074.796} C_VEL
LIN {X 0,Y 481.671,Z 335.482,A -85,B 0,C 180,E1 -7077.327,E2 -7077.327} C_VEL
LIN {X 0,Y 481.688,Z 335.483,A -85,B 0,C 180,E1 -7080.26,E2 -7080.26} C_VEL
LIN {X 0,Y 481.752,Z 335.471,A -85,B 0,C 180,E1 -7083.113,E2 -7083.113} C_VEL
LIN {X 0,Y 481.678,Z 335.489,A -85,B 0,C 180,E1 -7085.888,E2 -7085.888} C_VEL
LIN {X 0,Y 481.639,Z 335.488,A -85,B 0,C 180,E1 -7088.001,E2 -7088.001} C_VEL
LIN {X 0,Y 480.971,Z 335.57,A -85,B 0,C 180,E1 -7088.699,E2 -7088.699} C_VEL
LIN {X 0,Y 478.142,Z 335.929,A -85,B 0,C 180,E1 -7089.833,E2 -7089.833} C_VEL
LIN {X 0,Y 475.757,Z 336.222,A -85,B 0,C 180,E1 -7090.747,E2 -7090.747} C_VEL
LIN {X 0,Y 474.738,Z 336.348,A -85,B 0,C 180,E1 -7091.453,E2 -7091.453} C_VEL
LIN {X 0,Y 474.657,Z 336.36,A -85,B 0,C 180,E1 -7091.692,E2 -7091.692} C_VEL
LIN {X 0,Y 474.702,Z 336.35,A -85,B 0,C 180,E1 -7094.545,E2 -7094.545} C_VEL
LIN {X 0,Y 474.707,Z 336.353,A -85,B 0,C 180,E1 -7098.038,E2 -7098.038} C_VEL
LIN {X 0,Y 474.731,Z 336.352,A -85,B 0,C 180,E1 -7101.487,E2 -7101.487} C_VEL
LIN {X 0,Y 474.785,Z 336.342,A -85,B 0,C 180,E1 -7104.053,E2 -7104.053} C_VEL
LIN {X 0,Y 474.898,Z 336.332,A -85,B 0,C 180,E1 -7107.455,E2 -7107.455} C_VEL
LIN {X 0,Y 474.915,Z 336.325,A -85,B 0,C 180,E1 -7110,E2 -7110} C_VEL
LIN {X 0,Y 474.898,Z 336.325,A -85,B 0,C 180,E1 -7112.545,E2 -7112.545} C_VEL
LIN {X 0,Y 474.774,Z 336.343,A -85,B 0,C 180,E1 -7115.948,E2 -7115.948} C_VEL
LIN {X 0,Y 474.731,Z 336.346,A -85,B 0,C 180,E1 -7118.513,E2 -7118.513} C_VEL
LIN {X 0,Y 474.707,Z 336.35,A -85,B 0,C 180,E1 -7121.962,E2 -7121.962} C_VEL
LIN {X 0,Y 474.702,Z 336.356,A -85,B 0,C 180,E1 -7125.455,E2 -7125.455} C_VEL
LIN {X 0,Y 474.667,Z 336.358,A -85,B 0,C 180,E1 -7129.01,E2 -7129.01} C_VEL
LIN {X 0,Y 474.592,Z 336.365,A -85,B 0,C 180,E1 -7131.728,E2 -7131.728} C_VEL
LIN {X 0,Y 474.66,Z 336.355,A -85,B 0,C 180,E1 -7134.492,E2 -7134.492} C_VEL
LIN {X 0,Y 474.699,Z 336.356,A -85,B 0,C 180,E1 -7137.338,E2 -7137.338} C_VEL
LIN {X 0,Y 474.604,Z 336.366,A -85,B 0,C 180,E1 -7140.81,E2 -7140.81} C_VEL
LIN {X 0,Y 474.636,Z 336.357,A -85,B 0,C 180,E1 -7143.983,E2 -7143.983} C_VEL
LIN {X 0,Y 474.576,Z 336.372,A -85,B 0,C 180,E1 -7146.9,E2 -7146.9} C_VEL
LIN {X 0,Y 474.652,Z 336.358,A -85,B 0,C 180,E1 -7149.651,E2 -7149.651} C_VEL
LIN {X 0,Y 474.648,Z 336.364,A -85,B 0,C 180,E1 -7152.929,E2 -7152.929} C_VEL
LIN {X 0,Y 474.614,Z 336.365,A -85,B 0,C 180,E1 -7155.895,E2 -7155.895} C_VEL
LIN {X 0,Y 474.685,Z 336.473,A -85,B 0,C 180,E1 -7157.637,E2 -7157.637} C_VEL
LIN {X 0,Y 474.966,Z 337.768,A -85,B 0,C 180,E1 -7157.813,E2 -7157.813} C_VEL
LIN {X 0,Y 477.118,Z 345.772,A -85,B 0,C 180,E1 -7158.32,E2 -7158.32} C_VEL
LIN {X 0,Y 476.807,Z 356.481,A -85,B 0,C 180,E1 -7159.011,E2 -7159.011} C_VEL
LIN {X 0,Y 476.373,Z 367.178,A -85,B 0,C 180,E1 -7159.874,E2 -7159.874} C_VEL
LIN {X 0,Y 475.958,Z 378.09,A -85,B 0,C 180,E1 -7160.983,E2 -7160.983} C_VEL
LIN {X 0,Y 475.498,Z 387.464,A -85,B 0,C 180,E1 -7162.165,E2 -7162.165} C_VEL
LIN {X 0,Y 475.153,Z 395.781,A -85,B 0,C 180,E1 -7163.481,E2 -7163.481} C_VEL
LIN {X 0,Y 474.88,Z 402.224,A -85,B 0,C 180,E1 -7164.747,E2 -7164.747} C_VEL
LIN {X 0,Y 474.638,Z 407.382,A -85,B 0,C 180,E1 -7166.014,E2 -7166.014} C_VEL
LIN {X 0,Y 474.48,Z 411.251,A -85,B 0,C 180,E1 -7167.227,E2 -7167.227} C_VEL
LIN {X 0,Y 474.396,Z 414.832,A -85,B 0,C 180,E1 -7168.767,E2 -7168.767} C_VEL
LIN {X 0,Y 474.298,Z 416.384,A -85,B 0,C 180,E1 -7169.748,E2 -7169.748} C_VEL
LIN {X 0,Y 474.262,Z 417.57,A -85,B 0,C 180,E1 -7170.961,E2 -7170.961} C_VEL
LIN {X 0,Y 474.243,Z 417.917,A -85,B 0,C 180,E1 -7172.651,E2 -7172.651} C_VEL
LIN {X 0,Y 474.271,Z 417.398,A -85,B 0,C 180,E1 -7173.605,E2 -7173.605} C_VEL
LIN {X 0,Y 474.362,Z 416.286,A -85,B 0,C 180,E1 -7174.653,E2 -7174.653} C_VEL
LIN {X 0,Y 474.434,Z 414.93,A -85,B 0,C 180,E1 -7175.495,E2 -7175.495} C_VEL
LIN {X 0,Y 474.599,Z 412.418,A -85,B 0,C 180,E1 -7176.649,E2 -7176.649} C_VEL
LIN {X 0,Y 474.744,Z 408.999,A -85,B 0,C 180,E1 -7177.821,E2 -7177.821} C_VEL
LIN {X 0,Y 475.002,Z 403.79,A -85,B 0,C 180,E1 -7179.201,E2 -7179.201} C_VEL
LIN {X 0,Y 475.314,Z 397.112,A -85,B 0,C 180,E1 -7180.568,E2 -7180.568} C_VEL
LIN {X 0,Y 475.725,Z 388.763,A -85,B 0,C 180,E1 -7181.926,E2 -7181.926} C_VEL
LIN {X 0,Y 476.145,Z 379.962,A -85,B 0,C 180,E1 -7183.067,E2 -7183.067} C_VEL
LIN {X 0,Y 476.605,Z 369.406,A -85,B 0,C 180,E1 -7184.169,E2 -7184.169} C_VEL
LIN {X 0,Y 477.013,Z 358.73,A -85,B 0,C 180,E1 -7185.058,E2 -7185.058} C_VEL
LIN {X 0,Y 477.4,Z 346.815,A -85,B 0,C 180,E1 -7185.833,E2 -7185.833} C_VEL
LIN {X 0,Y 475.879,Z 340.737,A -85,B 0,C 180,E1 -7186.223,E2 -7186.223} C_VEL
LIN {X 0,Y 474.811,Z 337.093,A -85,B 0,C 180,E1 -7186.464,E2 -7186.464} C_VEL
LIN {X 0,Y 474.676,Z 336.379,A -85,B 0,C 180,E1 -7186.678,E2 -7186.678} C_VEL
LIN {X 0,Y 474.683,Z 336.358,A -85,B 0,C 180,E1 -7188.903,E2 -7188.903} C_VEL
LIN {X 0,Y 474.784,Z 336.342,A -85,B 0,C 180,E1 -7192.344,E2 -7192.344} C_VEL
LIN {X 0,Y 474.738,Z 336.351,A -85,B 0,C 180,E1 -7194.904,E2 -7194.904} C_VEL
LIN {X 0,Y 474.881,Z 336.335,A -85,B 0,C 180,E1 -7197.455,E2 -7197.455} C_VEL
LIN {X 0,Y 474.846,Z 336.336,A -85,B 0,C 180,E1 -7200.848,E2 -7200.848} C_VEL
LIN {X 0,Y 474.881,Z 336.329,A -85,B 0,C 180,E1 -7202.545,E2 -7202.545} C_VEL
LIN {X 0,Y 474.758,Z 336.345,A -85,B 0,C 180,E1 -7205.948,E2 -7205.948} C_VEL
LIN {X 0,Y 474.701,Z 336.351,A -85,B 0,C 180,E1 -7208.514,E2 -7208.514} C_VEL
LIN {X 0,Y 474.693,Z 336.351,A -85,B 0,C 180,E1 -7211.963,E2 -7211.963} C_VEL
LIN {X 0,Y 474.689,Z 336.356,A -85,B 0,C 180,E1 -7215.456,E2 -7215.456} C_VEL
LIN {X 0,Y 474.653,Z 336.363,A -85,B 0,C 180,E1 -7219.011,E2 -7219.011} C_VEL
LIN {X 0,Y 474.578,Z 336.367,A -85,B 0,C 180,E1 -7221.73,E2 -7221.73} C_VEL
LIN {X 0,Y 474.64,Z 336.359,A -85,B 0,C 180,E1 -7224.494,E2 -7224.494} C_VEL
LIN {X 0,Y 474.671,Z 336.358,A -85,B 0,C 180,E1 -7227.335,E2 -7227.335} C_VEL
LIN {X 0,Y 474.595,Z 336.369,A -85,B 0,C 180,E1 -7230.81,E2 -7230.81} C_VEL
LIN {X 0,Y 474.617,Z 336.365,A -85,B 0,C 180,E1 -7233.222,E2 -7233.222} C_VEL
LIN {X 0,Y 474.581,Z 336.369,A -85,B 0,C 180,E1 -7236.324,E2 -7236.324} C_VEL
LIN {X 0,Y 474.615,Z 336.364,A -85,B 0,C 180,E1 -7239.549,E2 -7239.549} C_VEL
LIN {X 0,Y 474.578,Z 336.37,A -85,B 0,C 180,E1 -7242.232,E2 -7242.232} C_VEL
LIN {X 0,Y 474.61,Z 336.366,A -85,B 0,C 180,E1 -7245.299,E2 -7245.299} C_VEL
LIN {X 0,Y 474.595,Z 336.367,A -85,B 0,C 180,E1 -7248.213,E2 -7248.213} C_VEL
LIN {X 0,Y 474.638,Z 336.577,A -85,B 0,C 180,E1 -7250.455,E2 -7250.455} C_VEL
LIN {X 0,Y 476.56,Z 346.459,A -85,B 0,C 180,E1 -7253.36,E2 -7253.36} C_VEL
LIN {X 0,Y 476.61,Z 350.864,A -85,B 0,C 180,E1 -7254.537,E2 -7254.537} C_VEL
LIN {X 0,Y 475.797,Z 366.211,A -85,B 0,C 180,E1 -7258.375,E2 -7258.375} C_VEL
LIN {X 0,Y 475.424,Z 379.465,A -85,B 0,C 180,E1 -7261.528,E2 -7261.528} C_VEL
LIN {X 0,Y 475.064,Z 393.889,A -85,B 0,C 180,E1 -7264.83,E2 -7264.83} C_VEL
LIN {X 0,Y 474.781,Z 407.348,A -85,B 0,C 180,E1 -7267.824,E2 -7267.824} C_VEL
LIN {X 0,Y 474.563,Z 420.827,A -85,B 0,C 180,E1 -7270.762,E2 -7270.762} C_VEL
LIN {X 0,Y 474.385,Z 434.235,A -85,B 0,C 180,E1 -7273.652,E2 -7273.652} C_VEL
LIN {X 0,Y 474.327,Z 439.561,A -85,B 0,C 180,E1 -7274.752,E2 -7274.752} C_VEL
LIN {X 0,Y 474.468,Z 441.603,A -85,B 0,C 180,E1 -7274.839,E2 -7274.839} C_VEL
LIN {X 0,Y 475.656,Z 456.608,A -85,B 0,C 180,E1 -7275.275,E2 -7275.275} C_VEL
LIN {X 0,Y 476.455,Z 465.578,A -85,B 0,C 180,E1 -7275.642,E2 -7275.642} C_VEL
LIN {X 0,Y 476.035,Z 477.545,A -85,B 0,C 180,E1 -7276.228,E2 -7276.228} C_VEL
LIN {X 0,Y 475.601,Z 489.333,A -85,B 0,C 180,E1 -7276.977,E2 -7276.977} C_VEL
LIN {X 0,Y 475.291,Z 499.031,A -85,B 0,C 180,E1 -7277.744,E2 -7277.744} C_VEL
LIN {X 0,Y 474.84,Z 508.891,A -85,B 0,C 180,E1 -7278.691,E2 -7278.691} C_VEL
LIN {X 0,Y 474.48,Z 518.076,A -85,B 0,C 180,E1 -7279.762,E2 -7279.762} C_VEL
LIN {X 0,Y 474.251,Z 527.107,A -85,B 0,C 180,E1 -7281.049,E2 -7281.049} C_VEL
LIN {X 0,Y 474.138,Z 534.351,A -85,B 0,C 180,E1 -7282.334,E2 -7282.334} C_VEL
LIN {X 0,Y 474.063,Z 540.23,A -85,B 0,C 180,E1 -7283.634,E2 -7283.634} C_VEL
LIN {X 0,Y 474.062,Z 544.738,A -85,B 0,C 180,E1 -7284.897,E2 -7284.897} C_VEL
LIN {X 0,Y 474.059,Z 547.164,A -85,B 0,C 180,E1 -7285.749,E2 -7285.749} C_VEL
LIN {X 0,Y 474.034,Z 549.14,A -85,B 0,C 180,E1 -7286.6,E2 -7286.6} C_VEL
LIN {X 0,Y 474.024,Z 550.63,A -85,B 0,C 180,E1 -7287.451,E2 -7287.451} C_VEL
LIN {X 0,Y 474.094,Z 552.382,A -85,B 0,C 180,E1 -7289.151,E2 -7289.151} C_VEL
LIN {X 0,Y 474.081,Z 552.638,A -85,B 0,C 180,E1 -7290,E2 -7290} C_VEL
LIN {X 0,Y 474.092,Z 552.444,A -85,B 0,C 180,E1 -7290.849,E2 -7290.849} C_VEL
LIN {X 0,Y 474,Z 550.839,A -85,B 0,C 180,E1 -7292.549,E2 -7292.549} C_VEL
LIN {X 0,Y 474.011,Z 549.41,A -85,B 0,C 180,E1 -7293.4,E2 -7293.4} C_VEL
LIN {X 0,Y 474,Z 546.412,A -85,B 0,C 180,E1 -7294.677,E2 -7294.677} C_VEL
LIN {X 0,Y 474.06,Z 542.343,A -85,B 0,C 180,E1 -7295.956,E2 -7295.956} C_VEL
LIN {X 0,Y 474.081,Z 536.055,A -85,B 0,C 180,E1 -7297.453,E2 -7297.453} C_VEL
LIN {X 0,Y 474.186,Z 529.214,A -85,B 0,C 180,E1 -7298.738,E2 -7298.738} C_VEL
LIN {X 0,Y 474.427,Z 520.721,A -85,B 0,C 180,E1 -7300.024,E2 -7300.024} C_VEL
LIN {X 0,Y 474.813,Z 512.02,A -85,B 0,C 180,E1 -7301.094,E2 -7301.094} C_VEL
LIN {X 0,Y 475.192,Z 503.693,A -85,B 0,C 180,E1 -7301.95,E2 -7301.95} C_VEL
LIN {X 0,Y 475.606,Z 492.225,A -85,B 0,C 180,E1 -7302.914,E2 -7302.914} C_VEL
LIN {X 0,Y 476.051,Z 481.048,A -85,B 0,C 180,E1 -7303.663,E2 -7303.663} C_VEL
LIN {X 0,Y 476.515,Z 468.534,A -85,B 0,C 180,E1 -7304.302,E2 -7304.302} C_VEL
LIN {X 0,Y 476.355,Z 462.219,A -85,B 0,C 180,E1 -7304.566,E2 -7304.566} C_VEL
LIN {X 0,Y 475.149,Z 449.902,A -85,B 0,C 180,E1 -7304.987,E2 -7304.987} C_VEL
LIN {X 0,Y 474.342,Z 441.838,A -85,B 0,C 180,E1 -7305.22,E2 -7305.22} C_VEL
LIN {X 0,Y 474.418,Z 435.495,A -85,B 0,C 180,E1 -7306.568,E2 -7306.568} C_VEL
LIN {X 0,Y 474.705,Z 422.48,A -85,B 0,C 180,E1 -7309.457,E2 -7309.457} C_VEL
LIN {X 0,Y 475.076,Z 408.457,A -85,B 0,C 180,E1 -7312.62,E2 -7312.62} C_VEL
LIN {X 0,Y 475.523,Z 394.112,A -85,B 0,C 180,E1 -7315.923,E2 -7315.923} C_VEL
LIN {X 0,Y 475.984,Z 380.37,A -85,B 0,C 180,E1 -7319.159,E2 -7319.159} C_VEL
LIN {X 0,Y 476.479,Z 368.339,A -85,B 0,C 180,E1 -7322.072,E2 -7322.072} C_VEL
LIN {X 0,Y 477.434,Z 352.799,A -85,B 0,C 180,E1 -7325.941,E2 -7325.941} C_VEL
LIN {X 0,Y 477.007,Z 348.228,A -85,B 0,C 180,E1 -7327.161,E2 -7327.161} C_VEL
LIN {X 0,Y 474.644,Z 336.464,A -85,B 0,C 180,E1 -7330.498,E2 -7330.498} C_VEL
LIN {X 0,Y 474.583,Z 336.372,A -85,B 0,C 180,E1 -7333.478,E2 -7333.478} C_VEL
LIN {X 0,Y 474.582,Z 336.367,A -85,B 0,C 180,E1 -7336.52,E2 -7336.52} C_VEL
LIN {X 0,Y 474.585,Z 336.372,A -85,B 0,C 180,E1 -7339.339,E2 -7339.339} C_VEL
LIN {X 0,Y 474.601,Z 336.365,A -85,B 0,C 180,E1 -7341.704,E2 -7341.704} C_VEL
LIN {X 0,Y 474.615,Z 336.362,A -85,B 0,C 180,E1 -7344.725,E2 -7344.725} C_VEL
LIN {X 0,Y 474.626,Z 336.361,A -85,B 0,C 180,E1 -7347.787,E2 -7347.787} C_VEL
LIN {X 0,Y 474.614,Z 336.364,A -85,B 0,C 180,E1 -7350.884,E2 -7350.884} C_VEL
LIN {X 0,Y 474.644,Z 336.359,A -85,B 0,C 180,E1 -7353.627,E2 -7353.627} C_VEL
LIN {X 0,Y 474.625,Z 336.361,A -85,B 0,C 180,E1 -7356.641,E2 -7356.641} C_VEL
LIN {X 0,Y 474.644,Z 336.357,A -85,B 0,C 180,E1 -7360.089,E2 -7360.089} C_VEL
LIN {X 0,Y 474.628,Z 336.363,A -85,B 0,C 180,E1 -7362.774,E2 -7362.774} C_VEL
LIN {X 0,Y 474.636,Z 336.36,A -85,B 0,C 180,E1 -7365.421,E2 -7365.421} C_VEL
LIN {X 0,Y 474.693,Z 336.35,A -85,B 0,C 180,E1 -7368.037,E2 -7368.037} C_VEL
LIN {X 0,Y 474.701,Z 336.351,A -85,B 0,C 180,E1 -7371.486,E2 -7371.486} C_VEL
LIN {X 0,Y 474.758,Z 336.343,A -85,B 0,C 180,E1 -7374.052,E2 -7374.052} C_VEL
LIN {X 0,Y 474.881,Z 336.328,A -85,B 0,C 180,E1 -7377.455,E2 -7377.455} C_VEL
LIN {X 0,Y 474.846,Z 336.339,A -85,B 0,C 180,E1 -7380.848,E2 -7380.848} C_VEL
LIN {X 0,Y 474.881,Z 336.332,A -85,B 0,C 180,E1 -7382.545,E2 -7382.545} C_VEL
LIN {X 0,Y 474.758,Z 336.343,A -85,B 0,C 180,E1 -7385.948,E2 -7385.948} C_VEL
LIN {X 0,Y 474.717,Z 336.353,A -85,B 0,C 180,E1 -7388.514,E2 -7388.514} C_VEL
LIN {X 0,Y 474.694,Z 336.351,A -85,B 0,C 180,E1 -7391.963,E2 -7391.963} C_VEL
LIN {X 0,Y 474.69,Z 336.351,A -85,B 0,C 180,E1 -7395.456,E2 -7395.456} C_VEL
LIN {X 0,Y 474.656,Z 336.357,A -85,B 0,C 180,E1 -7399.011,E2 -7399.011} C_VEL
LIN {X 0,Y 474.589,Z 336.364,A -85,B 0,C 180,E1 -7401.729,E2 -7401.729} C_VEL
LIN {X 0,Y 474.653,Z 336.363,A -85,B 0,C 180,E1 -7404.493,E2 -7404.493} C_VEL
LIN {X 0,Y 474.673,Z 336.353,A -85,B 0,C 180,E1 -7407.335,E2 -7407.335} C_VEL
LIN {X 0,Y 474.606,Z 336.368,A -85,B 0,C 180,E1 -7410.23,E2 -7410.23} C_VEL
LIN {X 0,Y 474.635,Z 336.358,A -85,B 0,C 180,E1 -7413.221,E2 -7413.221} C_VEL
LIN {X 0,Y 474.585,Z 336.372,A -85,B 0,C 180,E1 -7416.324,E2 -7416.324} C_VEL
LIN {X 0,Y 474.642,Z 336.358,A -85,B 0,C 180,E1 -7419.651,E2 -7419.651} C_VEL
LIN {X 0,Y 474.61,Z 336.361,A -85,B 0,C 180,E1 -7422.935,E2 -7422.935} C_VEL
LIN {X 0,Y 474.61,Z 336.365,A -85,B 0,C 180,E1 -7425.897,E2 -7425.897} C_VEL
LIN {X 0,Y 474.628,Z 336.358,A -85,B 0,C 180,E1 -7429.041,E2 -7429.041} C_VEL
LIN {X 0,Y 474.607,Z 336.365,A -85,B 0,C 180,E1 -7431.705,E2 -7431.705} C_VEL
LIN {X 0,Y 474.627,Z 336.359,A -85,B 0,C 180,E1 -7434.727,E2 -7434.727} C_VEL
LIN {X 0,Y 474.635,Z 336.363,A -85,B 0,C 180,E1 -7437.789,E2 -7437.789} C_VEL
LIN {X 0,Y 474.632,Z 336.358,A -85,B 0,C 180,E1 -7440.883,E2 -7440.883} C_VEL
LIN {X 0,Y 474.667,Z 336.358,A -85,B 0,C 180,E1 -7443.63,E2 -7443.63} C_VEL
LIN {X 0,Y 474.636,Z 336.358,A -85,B 0,C 180,E1 -7446.642,E2 -7446.642} C_VEL
LIN {X 0,Y 474.658,Z 336.359,A -85,B 0,C 180,E1 -7450.09,E2 -7450.09} C_VEL
LIN {X 0,Y 474.657,Z 336.36,A -85,B 0,C 180,E1 -7451.692,E2 -7451.692} C_VEL
LIN {X 0,Y 473.995,Z 336.447,A -85,B 0,C 180,E1 -7452.401,E2 -7452.401} C_VEL
LIN {X 0,Y 471.143,Z 336.802,A -85,B 0,C 180,E1 -7453.553,E2 -7453.553} C_VEL
LIN {X 0,Y 468.726,Z 337.098,A -85,B 0,C 180,E1 -7454.481,E2 -7454.481} C_VEL
LIN {X 0,Y 467.685,Z 337.225,A -85,B 0,C 180,E1 -7455.198,E2 -7455.198} C_VEL
LIN {X 0,Y 467.599,Z 337.235,A -85,B 0,C 180,E1 -7455.441,E2 -7455.441} C_VEL
LIN {X 0,Y 467.656,Z 337.227,A -85,B 0,C 180,E1 -7458.734,E2 -7458.734} C_VEL
LIN {X 0,Y 467.752,Z 337.217,A -85,B 0,C 180,E1 -7462.229,E2 -7462.229} C_VEL
LIN {X 0,Y 467.729,Z 337.218,A -85,B 0,C 180,E1 -7464.828,E2 -7464.828} C_VEL
LIN {X 0,Y 467.863,Z 337.207,A -85,B 0,C 180,E1 -7467.417,E2 -7467.417} C_VEL
LIN {X 0,Y 467.886,Z 337.201,A -85,B 0,C 180,E1 -7470,E2 -7470} C_VEL
LIN {X 0,Y 467.863,Z 337.201,A -85,B 0,C 180,E1 -7472.583,E2 -7472.583} C_VEL
LIN {X 0,Y 467.738,Z 337.218,A -85,B 0,C 180,E1 -7476.037,E2 -7476.037} C_VEL
LIN {X 0,Y 467.684,Z 337.224,A -85,B 0,C 180,E1 -7478.642,E2 -7478.642} C_VEL
LIN {X 0,Y 467.658,Z 337.227,A -85,B 0,C 180,E1 -7482.145,E2 -7482.145} C_VEL
LIN {X 0,Y 467.641,Z 337.232,A -85,B 0,C 180,E1 -7485.695,E2 -7485.695} C_VEL
LIN {X 0,Y 467.619,Z 337.234,A -85,B 0,C 180,E1 -7488.764,E2 -7488.764} C_VEL
LIN {X 0,Y 467.582,Z 337.244,A -85,B 0,C 180,E1 -7491.268,E2 -7491.268} C_VEL
LIN {X 0,Y 467.574,Z 337.238,A -85,B 0,C 180,E1 -7493.943,E2 -7493.943} C_VEL
LIN {X 0,Y 467.628,Z 337.234,A -85,B 0,C 180,E1 -7496.799,E2 -7496.799} C_VEL
LIN {X 0,Y 467.554,Z 337.241,A -85,B 0,C 180,E1 -7499.737,E2 -7499.737} C_VEL
LIN {X 0,Y 467.582,Z 337.24,A -85,B 0,C 180,E1 -7502.758,E2 -7502.758} C_VEL
LIN {X 0,Y 467.555,Z 337.24,A -85,B 0,C 180,E1 -7505.888,E2 -7505.888} C_VEL
LIN {X 0,Y 467.616,Z 337.239,A -85,B 0,C 180,E1 -7509.14,E2 -7509.14} C_VEL
LIN {X 0,Y 467.615,Z 337.238,A -85,B 0,C 180,E1 -7512.571,E2 -7512.571} C_VEL
LIN {X 0,Y 467.57,Z 337.243,A -85,B 0,C 180,E1 -7516.176,E2 -7516.176} C_VEL
LIN {X 0,Y 467.651,Z 337.408,A -85,B 0,C 180,E1 -7517.447,E2 -7517.447} C_VEL
LIN {X 0,Y 467.912,Z 338.631,A -85,B 0,C 180,E1 -7517.603,E2 -7517.603} C_VEL
LIN {X 0,Y 470.155,Z 346.708,A -85,B 0,C 180,E1 -7518.124,E2 -7518.124} C_VEL
LIN {X 0,Y 469.925,Z 357.707,A -85,B 0,C 180,E1 -7518.849,E2 -7518.849} C_VEL
LIN {X 0,Y 469.456,Z 368.82,A -85,B 0,C 180,E1 -7519.772,E2 -7519.772} C_VEL
LIN {X 0,Y 469.024,Z 379.301,A -85,B 0,C 180,E1 -7520.86,E2 -7520.86} C_VEL
LIN {X 0,Y 468.558,Z 388.553,A -85,B 0,C 180,E1 -7522.05,E2 -7522.05} C_VEL
LIN {X 0,Y 468.184,Z 396.751,A -85,B 0,C 180,E1 -7523.366,E2 -7523.366} C_VEL
LIN {X 0,Y 467.89,Z 403.364,A -85,B 0,C 180,E1 -7524.687,E2 -7524.687} C_VEL
LIN {X 0,Y 467.616,Z 409.312,A -85,B 0,C 180,E1 -7526.214,E2 -7526.214} C_VEL
LIN {X 0,Y 467.441,Z 413.846,A -85,B 0,C 180,E1 -7527.796,E2 -7527.796} C_VEL
LIN {X 0,Y 467.354,Z 416.714,A -85,B 0,C 180,E1 -7529.25,E2 -7529.25} C_VEL
LIN {X 0,Y 467.237,Z 418.436,A -85,B 0,C 180,E1 -7530.738,E2 -7530.738} C_VEL
LIN {X 0,Y 467.238,Z 418.935,A -85,B 0,C 180,E1 -7532.552,E2 -7532.552} C_VEL
LIN {X 0,Y 467.315,Z 417.961,A -85,B 0,C 180,E1 -7534.142,E2 -7534.142} C_VEL
LIN {X 0,Y 467.374,Z 416.701,A -85,B 0,C 180,E1 -7535.1,E2 -7535.1} C_VEL
LIN {X 0,Y 467.557,Z 414.021,A -85,B 0,C 180,E1 -7536.475,E2 -7536.475} C_VEL
LIN {X 0,Y 467.764,Z 409.958,A -85,B 0,C 180,E1 -7537.938,E2 -7537.938} C_VEL
LIN {X 0,Y 468.069,Z 404.719,A -85,B 0,C 180,E1 -7539.338,E2 -7539.338} C_VEL
LIN {X 0,Y 468.408,Z 398.029,A -85,B 0,C 180,E1 -7540.726,E2 -7540.726} C_VEL
LIN {X 0,Y 468.837,Z 389.664,A -85,B 0,C 180,E1 -7542.103,E2 -7542.103} C_VEL
LIN {X 0,Y 469.301,Z 380.751,A -85,B 0,C 180,E1 -7543.268,E2 -7543.268} C_VEL
LIN {X 0,Y 469.769,Z 370.235,A -85,B 0,C 180,E1 -7544.378,E2 -7544.378} C_VEL
LIN {X 0,Y 470.193,Z 359.487,A -85,B 0,C 180,E1 -7545.28,E2 -7545.28} C_VEL
LIN {X 0,Y 470.55,Z 347.575,A -85,B 0,C 180,E1 -7546.064,E2 -7546.064} C_VEL
LIN {X 0,Y 467.781,Z 338.025,A -85,B 0,C 180,E1 -7546.7,E2 -7546.7} C_VEL
LIN {X 0,Y 467.633,Z 337.26,A -85,B 0,C 180,E1 -7546.916,E2 -7546.916} C_VEL
LIN {X 0,Y 467.623,Z 337.238,A -85,B 0,C 180,E1 -7549.61,E2 -7549.61} C_VEL
LIN {X 0,Y 467.739,Z 337.22,A -85,B 0,C 180,E1 -7552.593,E2 -7552.593} C_VEL
LIN {X 0,Y 467.71,Z 337.226,A -85,B 0,C 180,E1 -7554.827,E2 -7554.827} C_VEL
LIN {X 0,Y 467.847,Z 337.21,A -85,B 0,C 180,E1 -7557.417,E2 -7557.417} C_VEL
LIN {X 0,Y 467.869,Z 337.204,A -85,B 0,C 180,E1 -7560,E2 -7560} C_VEL
LIN {X 0,Y 467.847,Z 337.206,A -85,B 0,C 180,E1 -7562.583,E2 -7562.583} C_VEL
LIN {X 0,Y 467.722,Z 337.221,A -85,B 0,C 180,E1 -7566.038,E2 -7566.038} C_VEL
LIN {X 0,Y 467.659,Z 337.229,A -85,B 0,C 180,E1 -7568.643,E2 -7568.643} C_VEL
LIN {X 0,Y 467.645,Z 337.229,A -85,B 0,C 180,E1 -7572.146,E2 -7572.146} C_VEL
LIN {X 0,Y 467.628,Z 337.234,A -85,B 0,C 180,E1 -7575.695,E2 -7575.695} C_VEL
LIN {X 0,Y 467.612,Z 337.238,A -85,B 0,C 180,E1 -7579.308,E2 -7579.308} C_VEL
LIN {X 0,Y 467.524,Z 337.245,A -85,B 0,C 180,E1 -7582.074,E2 -7582.074} C_VEL
LIN {X 0,Y 467.582,Z 337.243,A -85,B 0,C 180,E1 -7584.889,E2 -7584.889} C_VEL
LIN {X 0,Y 467.61,Z 337.235,A -85,B 0,C 180,E1 -7587.77,E2 -7587.77} C_VEL
LIN {X 0,Y 467.559,Z 337.244,A -85,B 0,C 180,E1 -7591.045,E2 -7591.045} C_VEL
LIN {X 0,Y 467.569,Z 337.241,A -85,B 0,C 180,E1 -7594.241,E2 -7594.241} C_VEL
LIN {X 0,Y 467.54,Z 337.248,A -85,B 0,C 180,E1 -7597.187,E2 -7597.187} C_VEL
LIN {X 0,Y 467.551,Z 337.245,A -85,B 0,C 180,E1 -7600.268,E2 -7600.268} C_VEL
LIN {X 0,Y 467.54,Z 337.245,A -85,B 0,C 180,E1 -7603.746,E2 -7603.746} C_VEL
LIN {X 0,Y 467.541,Z 337.246,A -85,B 0,C 180,E1 -7606.255,E2 -7606.255} C_VEL
LIN {X 0,Y 467.558,Z 337.246,A -85,B 0,C 180,E1 -7609.735,E2 -7609.735} C_VEL
